RoboDK station: kr30 cnc 040719 5.rdk

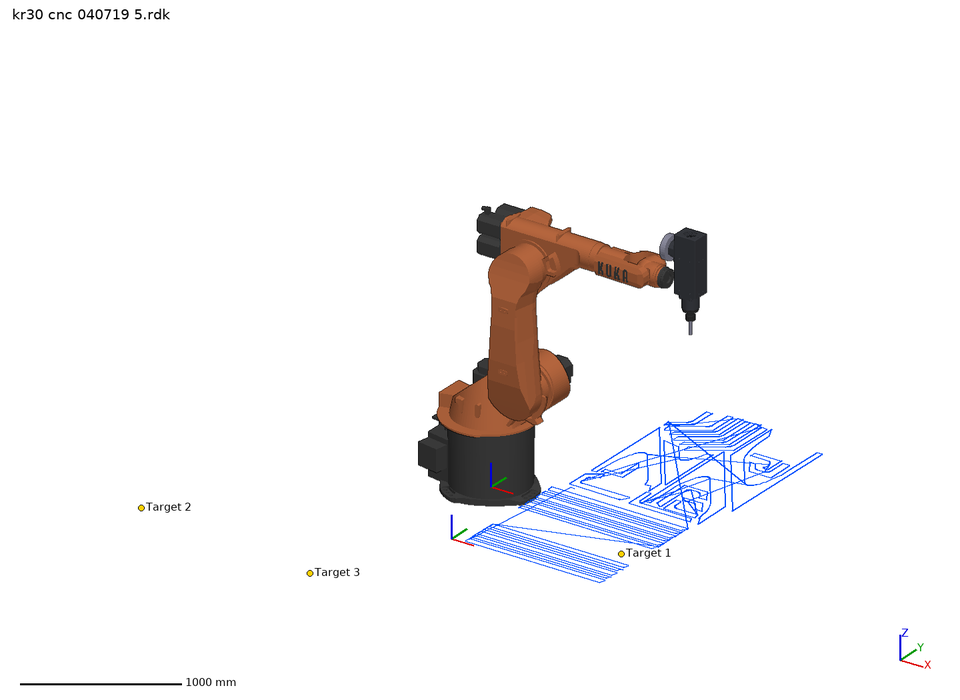
[picture v0: the station drawn from its stored meshes, robots at their saved joint values, targets as dots, program paths as lines]
Station kr30 cnc 040719 5. Poses are relative to the parent item; angles as X-Y-Z fixed-axis rotations.
  - frame KUKA KR 30 HA Base at (0, 0, 0) mm
    - robot KUKA KR 30 HA: 6 axes, payload 30 kg, reach 2033 mm, repeatability 0.05 mm, weight 665 kg
        modified DH rows (alpha deg, a mm, theta deg, d mm): 0, 0, 0, 815; -90, 350, 0, 0; 0, 850, -90, 0; -90, 145, 0, 820; 90, 0, 0, 0; -90, 0, 180, 170
        joint limits [-185, -135, -120, -350, -119, -350] to [185, 35, 158, 350, 119, 350]; home [0, -90, 90, 0, 0, 0]; saved at [0, -90, 90, 0, 0, 0]
      - tool 1/2" End Mill TCP, TCP at (337.71, -2.2, 160.57) mm, size 692.9 x 170 x 256 mm
    - frame Reference Rhino at (538.65, -1191.99, 269.68) mm
      - target Target 1 (Cartesian target) at (994.45, 406.4, 10) mm, rotated rx 0 ry 90 rz -60.43 deg; joints [16.304, -19.243, 71.371, -50.859, -63.853, 28.433] of KUKA KR 30 HA
      - target Target 2 (Cartesian target) at (-1810.84, -765.32, 10.08) mm, rotated rx 49.23 ry 89.99 rz -110.09 deg; joints [109.009, -5.295, 40.673, -64.339, -58.629, 47.297] of KUKA KR 30 HA
      - target Target 3 (Cartesian target) at (-425.52, -920.6, 10.08) mm, rotated rx 49.23 ry 89.99 rz -69.31 deg; joints [71.775, -8.447, 47.414, -59.408, -57.827, 42.008] of KUKA KR 30 HA
      - object RhinoPart at (0, 0, 0) mm
  - machining project RhinoPart Settings: C:/Users/Julian Ramirez.DESKTOP-JVDE542/Desktop/ELMER SHEET 1 TEST 3.nc | rotX(0) | rotY(270)*rotX(-65)
  - object box at (500, 500, 500) mm, size 250 x 250 x 250 mm, geometry from box.sld
  - program RhinoPart (549 instructions, listed below)
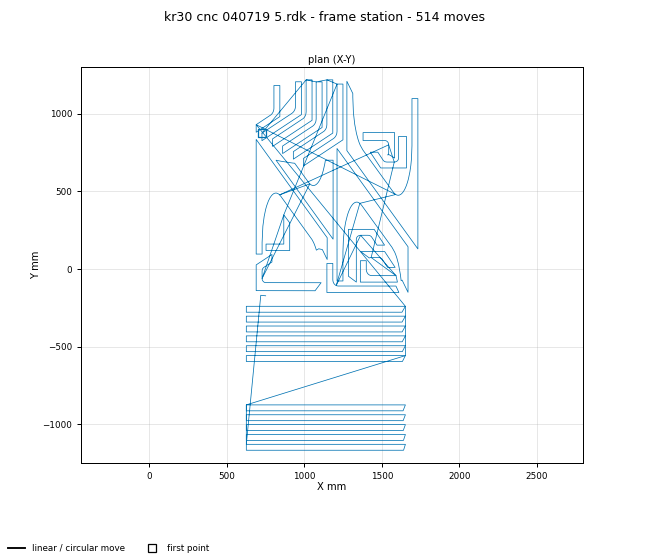
[picture p0: tool path of kr30 cnc 040719 5.rdk in frame station, 514 of 514 moves have a stored position in this frame; points joined in program order, loops and branches not executed]

--- program RhinoPart (robot KUKA KR 30 HA) ---
  Smooth(1)
  Set Ref.: Reference Rhino
  Set Tool: 1/2" End Mill TCP
  Show 1/2" End Mill TCP
  Set speed (2000.0 mm/s)
  MoveJ 1 to (189.6, 2067.69, 0) mm, rotated rx 0 ry 90 rz 29.57 deg; joints [-58.394, -46.833, 153.246, -29.84, -104.333, -8.083]
  MoveL 2 to (189.6, 2067.69, 0) mm, rotated rx 0 ry 90 rz 29.57 deg; joints [-58.394, -46.833, 153.246, -29.84, -104.333, -8.083]
  MoveL 3 to (189.6, 2067.69, 0) mm, rotated rx 0 ry 90 rz 29.57 deg; joints [-58.394, -46.833, 153.246, -29.84, -104.333, -8.083]
  Set speed (60.0 mm/s)
  MoveL 4 to (189.6, 2019.15, 0) mm, rotated rx 0 ry 90 rz 29.57 deg; joints [-56.567, -46.166, 155.923, -28.426, -107.53, -9.26]
  MoveL 5 to (443.6, 2187.03, 0) mm, rotated rx 0 ry 90 rz 29.57 deg; joints [-50.243, -46.091, 136.083, -20.671, -89.992, 0.003]
  MoveL 6 to (443.6, 2398.44, 0) mm, rotated rx 0 ry 90 rz 29.57 deg; joints [-56.43, -42.72, 123.102, -27.187, -81.428, 4.378]
  MoveL 7 to (405.5, 2398.44, 0) mm, rotated rx 0 ry 90 rz 29.57 deg; joints [-57.905, -43.217, 124.737, -28.597, -82.542, 4.047]
  MoveL 8 to (405.5, 2241.51, 0) mm, rotated rx 0 ry 90 rz 29.57 deg; joints [-53.573, -45.796, 134.651, -24.006, -88.954, 0.466]
  MoveL 9 to (405.1, 2234.61, 0) mm, rotated rx 0 ry 90 rz 29.57 deg; joints [-53.376, -45.887, 135.079, -23.806, -89.261, 0.326]
  MoveL 10 to (403.91, 2227.8, 0) mm, rotated rx 0 ry 90 rz 29.57 deg; joints [-53.213, -45.981, 135.535, -23.642, -89.591, 0.179]
  MoveL 11 to (401.94, 2221.18, 0) mm, rotated rx 0 ry 90 rz 29.57 deg; joints [-53.087, -46.077, 136.012, -23.515, -89.941, 0.026]
  MoveL 12 to (399.2, 2214.83, 0) mm, rotated rx 0 ry 90 rz 29.57 deg; joints [-53.001, -46.174, 136.507, -23.43, -90.305, -0.132]
  MoveL 13 to (395.69, 2208.84, 0) mm, rotated rx 0 ry 90 rz 29.57 deg; joints [-52.958, -46.27, 137.012, -23.388, -90.682, -0.295]
  MoveL 14 to (391.47, 2203.34, 0) mm, rotated rx 0 ry 90 rz 29.57 deg; joints [-52.961, -46.362, 137.518, -23.394, -91.061, -0.459]
  MoveL 15 to (386.58, 2198.44, 0) mm, rotated rx 0 ry 90 rz 29.57 deg; joints [-53.013, -46.45, 138.017, -23.449, -91.438, -0.624]
  MoveL 16 to (383.89, 2196.24, 0) mm, rotated rx 0 ry 90 rz 29.57 deg; joints [-53.057, -46.492, 138.263, -23.496, -91.624, -0.706]
  MoveL 17 to (381.06, 2194.23, 0) mm, rotated rx 0 ry 90 rz 29.57 deg; joints [-53.115, -46.533, 138.503, -23.556, -91.807, -0.788]
  MoveL 18 to (189.6, 2067.69, 0) mm, rotated rx 0 ry 90 rz 29.57 deg; joints [-58.394, -46.833, 153.246, -29.84, -104.333, -8.083]
  MoveL 19 to (474.07, 2410.87, 0) mm, rotated rx 0 ry 90 rz 29.57 deg; joints [-55.602, -42.027, 120.911, -26.461, -80.024, 4.928]
  Set speed (60.0 mm/s)
  MoveL 20 to (512.17, 2410.87, 0) mm, rotated rx 0 ry 90 rz 29.57 deg; joints [-54.221, -41.445, 119.132, -25.158, -78.824, 5.201]
  MoveL 21 to (512.17, 2150.2, 0) mm, rotated rx 0 ry 90 rz 29.57 deg; joints [-46.277, -45.815, 134.74, -16.708, -88.97, 0.309]
  MoveL 22 to (258.17, 1982.32, 0) mm, rotated rx 0 ry 90 rz 29.57 deg; joints [-51.067, -46.373, 155.224, -22.594, -107.496, -7.131]
  MoveL 23 to (258.17, 2030.85, 0) mm, rotated rx 0 ry 90 rz 29.57 deg; joints [-53.13, -46.929, 152.707, -24.376, -104.433, -6.444]
  MoveL 24 to (449.63, 2157.39, 0) mm, rotated rx 0 ry 90 rz 29.57 deg; joints [-48.975, -46.35, 137.45, -19.406, -91.038, -0.366]
  MoveL 25 to (455.15, 2161.61, 0) mm, rotated rx 0 ry 90 rz 29.57 deg; joints [-48.9, -46.258, 136.952, -19.33, -90.655, -0.23]
  MoveL 26 to (460.04, 2166.51, 0) mm, rotated rx 0 ry 90 rz 29.57 deg; joints [-48.876, -46.162, 136.446, -19.304, -90.268, -0.094]
  MoveL 27 to (464.26, 2172, 0) mm, rotated rx 0 ry 90 rz 29.57 deg; joints [-48.898, -46.062, 135.938, -19.327, -89.883, 0.041]
  MoveL 28 to (467.77, 2178, 0) mm, rotated rx 0 ry 90 rz 29.57 deg; joints [-48.966, -45.961, 135.435, -19.395, -89.504, 0.175]
  MoveL 29 to (470.51, 2184.35, 0) mm, rotated rx 0 ry 90 rz 29.57 deg; joints [-49.076, -45.859, 134.947, -19.506, -89.14, 0.305]
  MoveL 30 to (472.48, 2190.97, 0) mm, rotated rx 0 ry 90 rz 29.57 deg; joints [-49.223, -45.76, 134.48, -19.656, -88.795, 0.43]
  MoveL 31 to (474.07, 2204.68, 0) mm, rotated rx 0 ry 90 rz 29.57 deg; joints [-49.621, -45.572, 133.629, -20.06, -88.175, 0.666]
  MoveL 32 to (474.07, 2410.87, 0) mm, rotated rx 0 ry 90 rz 29.57 deg; joints [-55.602, -42.027, 120.911, -26.461, -80.024, 4.928]
  MoveL 33 to (538.73, 2397.73, 0) mm, rotated rx 0 ry 90 rz 29.57 deg; joints [-52.941, -41.304, 118.707, -23.882, -78.452, 5.065]
  Set speed (60.0 mm/s)
  MoveL 34 to (538.73, 2158.69, 0) mm, rotated rx 0 ry 90 rz 29.57 deg; joints [-45.6, -45.407, 132.909, -16.043, -87.598, 0.69]
  MoveL 35 to (537.14, 2144.98, 0) mm, rotated rx 0 ry 90 rz 29.57 deg; joints [-45.166, -45.593, 133.721, -15.602, -88.197, 0.503]
  MoveL 36 to (535.17, 2138.36, 0) mm, rotated rx 0 ry 90 rz 29.57 deg; joints [-44.997, -45.693, 134.174, -15.431, -88.536, 0.404]
  MoveL 37 to (532.43, 2132.01, 0) mm, rotated rx 0 ry 90 rz 29.57 deg; joints [-44.865, -45.797, 134.652, -15.296, -88.896, 0.302]
  MoveL 38 to (528.92, 2126.02, 0) mm, rotated rx 0 ry 90 rz 29.57 deg; joints [-44.772, -45.902, 135.149, -15.202, -89.274, 0.197]
  MoveL 39 to (524.7, 2120.53, 0) mm, rotated rx 0 ry 90 rz 29.57 deg; joints [-44.723, -46.006, 135.656, -15.152, -89.662, 0.091]
  MoveL 40 to (519.81, 2115.63, 0) mm, rotated rx 0 ry 90 rz 29.57 deg; joints [-44.721, -46.107, 136.165, -15.15, -90.056, -0.015]
  MoveL 41 to (514.29, 2111.41, 0) mm, rotated rx 0 ry 90 rz 29.57 deg; joints [-44.769, -46.205, 136.671, -15.197, -90.45, -0.122]
  MoveL 42 to (322.83, 1984.87, 0) mm, rotated rx 0 ry 90 rz 29.57 deg; joints [-47.793, -46.99, 152.328, -18.848, -104.552, -4.902]
  MoveL 43 to (322.83, 1936.34, 0) mm, rotated rx 0 ry 90 rz 29.57 deg; joints [-45.507, -46.523, 154.657, -16.723, -107.414, -5.138]
  MoveL 44 to (576.83, 2104.21, 0) mm, rotated rx 0 ry 90 rz 29.57 deg; joints [-42.246, -45.584, 133.683, -12.682, -88.145, 0.417]
  MoveL 45 to (576.83, 2397.73, 0) mm, rotated rx 0 ry 90 rz 29.57 deg; joints [-51.633, -40.652, 116.785, -22.658, -77.166, 5.298]
  MoveL 46 to (538.73, 2397.73, 0) mm, rotated rx 0 ry 90 rz 29.57 deg; joints [-52.941, -41.304, 118.707, -23.882, -78.452, 5.065]
  MoveL 47 to (607.72, 2410.87, 0) mm, rotated rx 0 ry 90 rz 29.57 deg; joints [-50.958, -39.788, 114.308, -22.115, -75.61, 5.767]
  Set speed (60.0 mm/s)
  MoveL 48 to (645.82, 2410.87, 0) mm, rotated rx 0 ry 90 rz 29.57 deg; joints [-49.734, -39.045, 112.237, -20.986, -74.25, 5.944]
  MoveL 49 to (645.82, 2068.09, 0) mm, rotated rx 0 ry 90 rz 29.57 deg; joints [-38.589, -45.07, 131.497, -9.034, -86.471, 0.561]
  MoveL 50 to (391.82, 1900.22, 0) mm, rotated rx 0 ry 90 rz 29.57 deg; joints [-40.437, -46.886, 152.953, -11.296, -105.771, -3.108]
  MoveL 51 to (391.82, 1948.75, 0) mm, rotated rx 0 ry 90 rz 29.57 deg; joints [-42.855, -47.182, 150.8, -13.654, -103.247, -3.186]
  MoveL 52 to (583.27, 2075.29, 0) mm, rotated rx 0 ry 90 rz 29.57 deg; joints [-40.908, -45.818, 134.752, -11.339, -88.955, 0.21]
  MoveL 53 to (588.8, 2079.51, 0) mm, rotated rx 0 ry 90 rz 29.57 deg; joints [-40.886, -45.707, 134.237, -11.318, -88.558, 0.289]
  MoveL 54 to (593.69, 2084.41, 0) mm, rotated rx 0 ry 90 rz 29.57 deg; joints [-40.912, -45.593, 133.723, -11.347, -88.166, 0.368]
  MoveL 55 to (597.91, 2089.9, 0) mm, rotated rx 0 ry 90 rz 29.57 deg; joints [-40.983, -45.478, 133.216, -11.42, -87.782, 0.448]
  MoveL 56 to (601.42, 2095.89, 0) mm, rotated rx 0 ry 90 rz 29.57 deg; joints [-41.096, -45.364, 132.723, -11.536, -87.412, 0.528]
  MoveL 57 to (604.16, 2102.24, 0) mm, rotated rx 0 ry 90 rz 29.57 deg; joints [-41.246, -45.253, 132.253, -11.69, -87.063, 0.608]
  MoveL 58 to (606.13, 2108.87, 0) mm, rotated rx 0 ry 90 rz 29.57 deg; joints [-41.431, -45.147, 131.813, -11.879, -86.737, 0.686]
  MoveL 59 to (607.72, 2122.58, 0) mm, rotated rx 0 ry 90 rz 29.57 deg; joints [-41.89, -44.955, 131.034, -12.346, -86.17, 0.838]
  MoveL 60 to (607.72, 2410.87, 0) mm, rotated rx 0 ry 90 rz 29.57 deg; joints [-50.958, -39.788, 114.308, -22.115, -75.61, 5.767]
  MoveL 61 to (673.1, 2383.75, 0) mm, rotated rx 0 ry 90 rz 29.57 deg; joints [-48.146, -39.124, 112.454, -19.33, -74.222, 5.448]
  Set speed (60.0 mm/s)
  MoveL 62 to (673.1, 2079.03, 0) mm, rotated rx 0 ry 90 rz 29.57 deg; joints [-38.176, -44.522, 129.354, -8.639, -84.89, 0.775]
  MoveL 63 to (671.52, 2065.32, 0) mm, rotated rx 0 ry 90 rz 29.57 deg; joints [-37.693, -44.715, 130.093, -8.148, -85.424, 0.654]
  MoveL 64 to (669.55, 2058.7, 0) mm, rotated rx 0 ry 90 rz 29.57 deg; joints [-37.494, -44.825, 130.519, -7.945, -85.735, 0.595]
  MoveL 65 to (666.8, 2052.35, 0) mm, rotated rx 0 ry 90 rz 29.57 deg; joints [-37.327, -44.941, 130.977, -7.773, -86.073, 0.536]
  MoveL 66 to (663.29, 2046.36, 0) mm, rotated rx 0 ry 90 rz 29.57 deg; joints [-37.195, -45.061, 131.463, -7.638, -86.434, 0.478]
  MoveL 67 to (659.07, 2040.86, 0) mm, rotated rx 0 ry 90 rz 29.57 deg; joints [-37.103, -45.184, 131.967, -7.543, -86.811, 0.422]
  MoveL 68 to (654.18, 2035.96, 0) mm, rotated rx 0 ry 90 rz 29.57 deg; joints [-37.055, -45.308, 132.483, -7.492, -87.2, 0.368]
  MoveL 69 to (648.66, 2031.74, 0) mm, rotated rx 0 ry 90 rz 29.57 deg; joints [-37.053, -45.429, 133.004, -7.488, -87.596, 0.316]
  MoveL 70 to (457.2, 1905.21, 0) mm, rotated rx 0 ry 90 rz 29.57 deg; joints [-37.971, -47.293, 149.341, -8.586, -101.917, -1.786]
  MoveL 71 to (457.2, 1856.67, 0) mm, rotated rx 0 ry 90 rz 29.57 deg; joints [-35.445, -47.128, 151.299, -6.056, -104.096, -1.48]
  MoveL 72 to (711.2, 2024.55, 0) mm, rotated rx 0 ry 90 rz 29.57 deg; joints [-34.93, -44.559, 129.495, -5.379, -84.958, 0.474]
  MoveL 73 to (711.2, 2383.75, 0) mm, rotated rx 0 ry 90 rz 29.57 deg; joints [-46.992, -38.31, 110.233, -18.266, -72.779, 5.581]
  MoveL 74 to (673.1, 2383.75, 0) mm, rotated rx 0 ry 90 rz 29.57 deg; joints [-48.146, -39.124, 112.454, -19.33, -74.222, 5.448]
  MoveL 75 to (330.2, 1541.24, 0) mm, rotated rx 180 ry 60 rz -150.43 deg; joints [-20.955, -60.967, 157.047, 8.164, -66.015, 0.995]
  Set speed (60.0 mm/s)
  MoveL 76 to (365.54, 1493.75, 0) mm, rotated rx -180 ry 60 rz -150.43 deg; joints [-17.055, -60.795, 155.789, 11.964, -64.88, 1.194]
  MoveL 77 to (368.3, 1490.21, 0) mm, rotated rx -180 ry 60 rz -150.43 deg; joints [-16.768, -60.778, 155.676, 12.248, -64.781, 1.198]
  MoveL 78 to (368.3, 1311.73, 0) mm, rotated rx -180 ry 60 rz -150.43 deg; joints [-4.531, -61.072, 157.995, 23.596, -66.311, 3.194]
  MoveL 79 to (215.9, 1311.73, 0) mm, rotated rx -180 ry 30 rz -150.43 deg; joints [-12.047, -59.926, 152.531, 16.276, -32.492, 1.46]
  MoveL 80 to (215.9, 1353.22, 0) mm, rotated rx -180 ry 40 rz -150.43 deg; joints [-13.186, -62.573, 157.529, 14.92, -44.772, 1.983]
  MoveL 81 to (330.2, 1353.22, 0) mm, rotated rx -180 ry 50 rz -150.43 deg; joints [-9.855, -62.245, 155.167, 18.943, -52.758, 1.238]
  MoveL 82 to (330.2, 1541.24, 0) mm, rotated rx -180 ry 60 rz -150.43 deg; joints [-20.955, -60.967, 157.047, 8.164, -66.015, 0.995]
  MoveL 83 to (190.5, 1131.98, 0) mm, rotated rx -180 ry 30 rz -150.43 deg; joints [-0.319, -60.475, 155.694, 25.458, -34.639, 4.485]
  Set speed (60.0 mm/s)
  MoveL 84 to (190.5, 1180.23, 0) mm, rotated rx -180 ry 30 rz -150.43 deg; joints [-3.61, -60.458, 155.578, 22.631, -34.669, 3.938]
  MoveL 85 to (191.3, 1187.11, 0) mm, rotated rx -180 ry 30 rz -150.43 deg; joints [-4.074, -60.445, 155.489, 22.265, -34.615, 3.82]
  MoveL 86 to (192.29, 1190.42, 0) mm, rotated rx -180 ry 30 rz -150.43 deg; joints [-4.294, -60.432, 155.403, 22.112, -34.554, 3.74]
  MoveL 87 to (193.65, 1193.58, 0) mm, rotated rx -180 ry 30 rz -150.43 deg; joints [-4.501, -60.415, 155.291, 21.982, -34.472, 3.648]
  MoveL 88 to (195.39, 1196.56, 0) mm, rotated rx -180 ry 30 rz -150.43 deg; joints [-4.692, -60.394, 155.152, 21.877, -34.369, 3.544]
  MoveL 89 to (197.49, 1199.29, 0) mm, rotated rx -180 ry 30 rz -150.43 deg; joints [-4.865, -60.369, 154.99, 21.799, -34.247, 3.43]
  MoveL 90 to (199.93, 1201.75, 0) mm, rotated rx -180 ry 30 rz -150.43 deg; joints [-5.016, -60.339, 154.803, 21.751, -34.106, 3.307]
  MoveL 91 to (202.72, 1203.88, 0) mm, rotated rx -180 ry 30 rz -150.43 deg; joints [-5.142, -60.305, 154.595, 21.735, -33.947, 3.175]
  MoveL 92 to (254, 1237.77, 0) mm, rotated rx -180 ry 40 rz -150.43 deg; joints [-4.845, -62.336, 156.153, 22.996, -43.491, 2.319]
  MoveL 93 to (254, 1286.3, 0) mm, rotated rx -180 ry 40 rz -150.43 deg; joints [-8.144, -62.263, 155.766, 20.032, -43.277, 1.866]
  MoveL 94 to (152.4, 1219.15, 0) mm, rotated rx -180 ry 30 rz -150.43 deg; joints [-6.544, -60.743, 157.989, 19.072, -36.768, 4.728]
  MoveL 95 to (152.4, 1053.37, 0) mm, rotated rx -180 ry 20 rz -150.43 deg; joints [2.369, -56.869, 153.192, 24.779, -25.576, 7.756]
  MoveL 96 to (520.7, 1053.37, 0) mm, rotated rx 0 ry 90 rz 29.57 deg; joints [21.258, -46.671, 154.029, 52.131, -100.861, 13.621]
  MoveL 97 to (523.39, 1053.29, 0) mm, rotated rx 0 ry 90 rz 29.57 deg; joints [21.196, -46.708, 153.862, 52.038, -100.751, 13.446]
  MoveL 98 to (526.09, 1053.06, 0) mm, rotated rx 0 ry 90 rz 29.57 deg; joints [21.144, -46.744, 153.691, 51.956, -100.635, 13.271]
  MoveL 99 to (528.75, 1052.67, 0) mm, rotated rx 0 ry 90 rz 29.57 deg; joints [21.102, -46.78, 153.518, 51.884, -100.516, 13.096]
  MoveL 100 to (531.38, 1052.13, 0) mm, rotated rx 0 ry 90 rz 29.57 deg; joints [21.072, -46.814, 153.343, 51.824, -100.394, 12.924]
  MoveL 101 to (570.41, 1104.33, 0) mm, rotated rx 0 ry 90 rz 29.57 deg; joints [16.876, -47.035, 152.019, 47.436, -100.261, 10.977]
  MoveL 102 to (215.9, 1104.33, 0) mm, rotated rx 180 ry 30 rz -150.43 deg; joints [1.524, -60.184, 153.886, 28.122, -33.22, 3.49]
  MoveL 103 to (210.71, 1104.91, 0) mm, rotated rx -180 ry 30 rz -150.43 deg; joints [1.494, -60.248, 154.253, 27.879, -33.489, 3.745]
  MoveL 104 to (208.23, 1105.62, 0) mm, rotated rx -180 ry 30 rz -150.43 deg; joints [1.451, -60.278, 154.429, 27.738, -33.619, 3.864]
  MoveL 105 to (205.85, 1106.58, 0) mm, rotated rx -180 ry 30 rz -150.43 deg; joints [1.391, -60.306, 154.599, 27.585, -33.746, 3.975]
  MoveL 106 to (203.58, 1107.8, 0) mm, rotated rx -180 ry 30 rz -150.43 deg; joints [1.313, -60.332, 154.76, 27.421, -33.869, 4.078]
  MoveL 107 to (201.44, 1109.25, 0) mm, rotated rx -180 ry 30 rz -150.43 deg; joints [1.218, -60.357, 154.913, 27.25, -33.986, 4.171]
  MoveL 108 to (199.45, 1110.91, 0) mm, rotated rx -180 ry 30 rz -150.43 deg; joints [1.109, -60.379, 155.056, 27.071, -34.097, 4.255]
  MoveL 109 to (197.61, 1112.79, 0) mm, rotated rx -180 ry 30 rz -150.43 deg; joints [0.984, -60.4, 155.187, 26.886, -34.201, 4.329]
  MoveL 110 to (195.97, 1114.84, 0) mm, rotated rx -180 ry 30 rz -150.43 deg; joints [0.847, -60.418, 155.305, 26.698, -34.295, 4.39]
  MoveL 111 to (194.53, 1117.03, 0) mm, rotated rx -180 ry 30 rz -150.43 deg; joints [0.7, -60.433, 155.407, 26.511, -34.379, 4.44]
  MoveL 112 to (192.31, 1121.74, 0) mm, rotated rx 180 ry 30 rz -150.43 deg; joints [0.38, -60.456, 155.567, 26.141, -34.513, 4.502]
  MoveL 113 to (190.96, 1126.77, 0) mm, rotated rx -180 ry 30 rz -150.43 deg; joints [0.037, -60.47, 155.663, 25.787, -34.601, 4.516]
  MoveL 114 to (190.5, 1131.98, 0) mm, rotated rx -180 ry 30 rz -150.43 deg; joints [-0.319, -60.475, 155.694, 25.458, -34.639, 4.485]
  MoveL 115 to (497.79, 1740.88, 0) mm, rotated rx -180 ry 80 rz -150.43 deg; joints [-27.553, -52.725, 149.919, 1.99, -87.19, 0.253]
  Set speed (60.0 mm/s)
  MoveL 116 to (502.27, 1737.01, 0) mm, rotated rx 0 ry 90 rz 29.57 deg; joints [-27.028, -46.901, 152.872, 2.646, -105.955, 0.728]
  MoveL 117 to (506.69, 1734.05, 0) mm, rotated rx 0 ry 90 rz 29.57 deg; joints [-26.714, -46.93, 152.699, 2.969, -105.749, 0.807]
  MoveL 118 to (511.04, 1731.95, 0) mm, rotated rx 0 ry 90 rz 29.57 deg; joints [-26.455, -46.962, 152.503, 3.234, -105.517, 0.866]
  MoveL 119 to (515.31, 1730.65, 0) mm, rotated rx 0 ry 90 rz 29.57 deg; joints [-26.249, -46.996, 152.287, 3.444, -105.264, 0.908]
  MoveL 120 to (519.5, 1730.11, 0) mm, rotated rx 0 ry 90 rz 29.57 deg; joints [-26.093, -47.031, 152.052, 3.601, -104.993, 0.933]
  MoveL 121 to (523.61, 1730.27, 0) mm, rotated rx 0 ry 90 rz 29.57 deg; joints [-25.983, -47.065, 151.801, 3.711, -104.706, 0.943]
  MoveL 122 to (527.62, 1731.09, 0) mm, rotated rx 0 ry 90 rz 29.57 deg; joints [-25.915, -47.1, 151.536, 3.775, -104.406, 0.941]
  MoveL 123 to (531.52, 1732.52, 0) mm, rotated rx 0 ry 90 rz 29.57 deg; joints [-25.887, -47.133, 151.259, 3.799, -104.097, 0.926]
  MoveL 124 to (535.31, 1734.5, 0) mm, rotated rx 0 ry 90 rz 29.57 deg; joints [-25.896, -47.164, 150.972, 3.785, -103.779, 0.903]
  MoveL 125 to (538.98, 1736.99, 0) mm, rotated rx 0 ry 90 rz 29.57 deg; joints [-25.937, -47.194, 150.677, 3.737, -103.455, 0.871]
  MoveL 126 to (542.53, 1739.94, 0) mm, rotated rx 0 ry 90 rz 29.57 deg; joints [-26.009, -47.221, 150.375, 3.659, -103.128, 0.832]
  MoveL 127 to (545.93, 1743.29, 0) mm, rotated rx 0 ry 90 rz 29.57 deg; joints [-26.107, -47.246, 150.069, 3.553, -102.799, 0.788]
  MoveL 128 to (552.31, 1751, 0) mm, rotated rx 0 ry 90 rz 29.57 deg; joints [-26.37, -47.287, 149.45, 3.274, -102.144, 0.69]
  MoveL 129 to (557.85, 1759.34, 0) mm, rotated rx 0 ry 90 rz 29.57 deg; joints [-26.688, -47.315, 148.86, 2.943, -101.53, 0.589]
  MoveL 130 to (562.91, 1768.41, 0) mm, rotated rx 0 ry 90 rz 29.57 deg; joints [-27.054, -47.334, 148.271, 2.564, -100.927, 0.486]
  MoveL 131 to (567.51, 1777.97, 0) mm, rotated rx 0 ry 90 rz 29.57 deg; joints [-27.453, -47.343, 147.691, 2.154, -100.341, 0.387]
  MoveL 132 to (576.13, 1799.75, 0) mm, rotated rx 0 ry 90 rz 29.57 deg; joints [-28.39, -47.334, 146.463, 1.197, -99.127, 0.19]
  MoveL 133 to (584.02, 1825.23, 0) mm, rotated rx 0 ry 90 rz 29.57 deg; joints [-29.506, -47.284, 145.126, 0.067, -97.843, 0.009]
  MoveL 134 to (593.39, 1865.46, 0) mm, rotated rx 0 ry 90 rz 29.57 deg; joints [-31.271, -47.139, 143.131, -1.709, -95.989, -0.178]
  MoveL 135 to (598.13, 1892.37, 0) mm, rotated rx 0 ry 90 rz 29.57 deg; joints [-32.442, -47.005, 141.839, -2.881, -94.828, -0.243]
  MoveL 136 to (609.6, 1893.44, 0) mm, rotated rx 0 ry 90 rz 29.57 deg; joints [-32.146, -46.916, 141.107, -2.581, -94.186, -0.189]
  MoveL 137 to (647.7, 1893.44, 0) mm, rotated rx 0 ry 90 rz 29.57 deg; joints [-31.037, -46.577, 138.772, -1.467, -92.195, -0.056]
  MoveL 138 to (647.7, 1384.85, 0) mm, rotated rx 0 ry 90 rz 29.57 deg; joints [-2.018, -47.297, 149.263, 28.074, -100.592, 5.599]
  MoveL 139 to (280.37, 1893.44, 0) mm, rotated rx -180 ry 80 rz -150.43 deg; joints [-44.299, -52.692, 155.935, -14.517, -92.817, -3.343]
  MoveL 140 to (309.91, 1887.14, 0) mm, rotated rx 0 ry 90 rz 29.57 deg; joints [-43.636, -45.609, 157.481, -15.108, -111.184, -5.572]
  MoveL 141 to (385.37, 1875.31, 0) mm, rotated rx 0 ry 90 rz 29.57 deg; joints [-39.408, -46.602, 154.332, -10.317, -107.461, -3.126]
  MoveL 142 to (400.34, 1873.88, 0) mm, rotated rx 0 ry 90 rz 29.57 deg; joints [-38.679, -46.757, 153.628, -9.509, -106.651, -2.748]
  MoveL 143 to (488.7, 1751.54, 0) mm, rotated rx 0 ry 90 rz 29.57 deg; joints [-28.332, -46.837, 153.22, 1.292, -106.379, 0.364]
  MoveL 144 to (493.27, 1745.7, 0) mm, rotated rx 0 ry 90 rz 29.57 deg; joints [-27.835, -46.853, 153.135, 1.809, -106.274, 0.507]
  MoveL 145 to (497.79, 1740.88, 0) mm, rotated rx 0 ry 90 rz 29.57 deg; joints [-27.401, -46.875, 153.018, 2.26, -106.131, 0.628]
  MoveL 146 to (303.35, 1670.14, 0) mm, rotated rx -180 ry 60 rz -150.43 deg; joints [-29.742, -60.649, 154.872, -0.164, -64.222, -0.014]
  Set speed (60.0 mm/s)
  MoveL 147 to (307.39, 1665.7, 0) mm, rotated rx -180 ry 60 rz -150.43 deg; joints [-29.348, -60.634, 154.778, 0.215, -64.144, 0.018]
  MoveL 148 to (311.4, 1660.54, 0) mm, rotated rx -180 ry 60 rz -150.43 deg; joints [-28.914, -60.622, 154.708, 0.633, -64.086, 0.052]
  MoveL 149 to (511.79, 1382.48, 0) mm, rotated rx -180 ry 80 rz -150.43 deg; joints [-4.246, -52.699, 155.869, 24.929, -91.933, 5.596]
  MoveL 150 to (516.77, 1373.81, 0) mm, rotated rx 0 ry 90 rz 29.57 deg; joints [-1.538, -45.433, 157.901, 29.951, -109.714, 11]
  MoveL 151 to (521.42, 1364.56, 0) mm, rotated rx 0 ry 90 rz 29.57 deg; joints [-0.842, -45.553, 157.618, 30.603, -109.233, 11.025]
  MoveL 152 to (525.76, 1354.87, 0) mm, rotated rx 0 ry 90 rz 29.57 deg; joints [-0.122, -45.662, 157.346, 31.284, -108.769, 11.062]
  MoveL 153 to (533.5, 1334.64, 0) mm, rotated rx 0 ry 90 rz 29.57 deg; joints [1.359, -45.856, 156.837, 32.691, -107.887, 11.151]
  MoveL 154 to (540.04, 1314.08, 0) mm, rotated rx 0 ry 90 rz 29.57 deg; joints [2.836, -46.02, 156.369, 34.1, -107.072, 11.242]
  MoveL 155 to (555.23, 1322.96, 0) mm, rotated rx 0 ry 90 rz 29.57 deg; joints [2.152, -46.319, 155.412, 33.192, -106.155, 10.316]
  MoveL 156 to (561.07, 1321.73, 0) mm, rotated rx 0 ry 90 rz 29.57 deg; joints [2.223, -46.426, 155.029, 33.188, -105.732, 10.057]
  MoveL 157 to (578.58, 1317.86, 0) mm, rotated rx 0 ry 90 rz 29.57 deg; joints [2.444, -46.706, 153.873, 33.201, -104.494, 9.301]
  MoveL 158 to (609.6, 1253.88, 0) mm, rotated rx 0 ry 90 rz 29.57 deg; joints [6.592, -47.106, 151.485, 37.037, -101.566, 8.603]
  MoveL 159 to (609.6, 1394.22, 0) mm, rotated rx 0 ry 90 rz 29.57 deg; joints [-2.73, -47.065, 151.802, 27.621, -103.119, 6.773]
  MoveL 160 to (152.4, 2027.23, 0) mm, rotated rx 180 ry 70 rz -150.43 deg; joints [-54.922, -56.98, 150.659, -24.834, -73.332, -1.643]
  MoveL 161 to (152.4, 1288.87, 0) mm, rotated rx 180 ry 20 rz -150.43 deg; joints [-12.956, -56.684, 151.653, 13.483, -24.8, 3.385]
  MoveL 162 to (190.5, 1288.87, 0) mm, rotated rx -180 ry 30 rz -150.43 deg; joints [-10.903, -60.308, 154.611, 16.586, -34.102, 2.455]
  MoveL 163 to (190.5, 1362.91, 0) mm, rotated rx -180 ry 30 rz -150.43 deg; joints [-15.691, -60.096, 153.409, 12.646, -33.224, 1.45]
  MoveL 164 to (195.47, 1468.11, 0) mm, rotated rx -180 ry 40 rz -150.43 deg; joints [-21.259, -62.401, 156.508, 7.678, -44.067, 0.853]
  MoveL 165 to (203.82, 1530.87, 0) mm, rotated rx -180 ry 40 rz -150.43 deg; joints [-24.948, -61.945, 154.226, 4.417, -42.274, 0.273]
  MoveL 166 to (213.36, 1576.46, 0) mm, rotated rx -180 ry 40 rz -150.43 deg; joints [-27.349, -61.467, 152.189, 2.19, -40.722, 0.043]
  MoveL 167 to (219.68, 1599.23, 0) mm, rotated rx -180 ry 50 rz -150.43 deg; joints [-28.331, -62.572, 156.878, 1.17, -54.305, 0.115]
  MoveL 168 to (227.14, 1620.99, 0) mm, rotated rx -180 ry 50 rz -150.43 deg; joints [-29.394, -62.348, 155.679, 0.17, -53.331, 0.013]
  MoveL 169 to (231.16, 1630.88, 0) mm, rotated rx -180 ry 50 rz -150.43 deg; joints [-29.842, -62.228, 155.087, -0.259, -52.859, -0.017]
  MoveL 170 to (235.75, 1640.83, 0) mm, rotated rx -180 ry 50 rz -150.43 deg; joints [-30.265, -62.093, 154.453, -0.671, -52.36, -0.036]
  MoveL 171 to (240.92, 1650.5, 0) mm, rotated rx -180 ry 50 rz -150.43 deg; joints [-30.644, -61.945, 153.79, -1.045, -51.845, -0.044]
  MoveL 172 to (246.67, 1659.52, 0) mm, rotated rx -180 ry 50 rz -150.43 deg; joints [-30.959, -61.786, 153.111, -1.362, -51.324, -0.041]
  MoveL 173 to (250.51, 1664.62, 0) mm, rotated rx -180 ry 50 rz -150.43 deg; joints [-31.115, -61.684, 152.689, -1.521, -51.005, -0.035]
  MoveL 174 to (254.42, 1669.07, 0) mm, rotated rx -180 ry 60 rz -150.43 deg; joints [-31.397, -61.058, 157.861, -1.72, -66.799, -0.235]
  MoveL 175 to (258.37, 1672.87, 0) mm, rotated rx -180 ry 60 rz -150.43 deg; joints [-31.48, -61.018, 157.487, -1.803, -66.466, -0.235]
  MoveL 176 to (262.38, 1676.02, 0) mm, rotated rx -180 ry 60 rz -150.43 deg; joints [-31.522, -60.977, 157.134, -1.847, -66.154, -0.229]
  MoveL 177 to (266.41, 1678.5, 0) mm, rotated rx -180 ry 60 rz -150.43 deg; joints [-31.522, -60.936, 156.803, -1.851, -65.864, -0.218]
  MoveL 178 to (270.48, 1680.31, 0) mm, rotated rx -180 ry 60 rz -150.43 deg; joints [-31.482, -60.896, 156.494, -1.817, -65.595, -0.205]
  MoveL 179 to (274.58, 1681.45, 0) mm, rotated rx -180 ry 60 rz -150.43 deg; joints [-31.402, -60.856, 156.208, -1.744, -65.349, -0.188]
  MoveL 180 to (278.69, 1681.92, 0) mm, rotated rx -180 ry 60 rz -150.43 deg; joints [-31.282, -60.818, 155.945, -1.633, -65.124, -0.168]
  MoveL 181 to (282.81, 1681.7, 0) mm, rotated rx -180 ry 60 rz -150.43 deg; joints [-31.123, -60.783, 155.705, -1.483, -64.921, -0.147]
  MoveL 182 to (286.94, 1680.79, 0) mm, rotated rx -180 ry 60 rz -150.43 deg; joints [-30.925, -60.75, 155.49, -1.296, -64.739, -0.124]
  MoveL 183 to (291.06, 1679.18, 0) mm, rotated rx -180 ry 60 rz -150.43 deg; joints [-30.688, -60.719, 155.299, -1.07, -64.578, -0.099]
  MoveL 184 to (295.17, 1676.87, 0) mm, rotated rx -180 ry 60 rz -150.43 deg; joints [-30.411, -60.693, 155.132, -0.806, -64.439, -0.072]
  MoveL 185 to (299.27, 1673.86, 0) mm, rotated rx -180 ry 60 rz -150.43 deg; joints [-30.096, -60.669, 154.99, -0.504, -64.32, -0.044]
  MoveL 186 to (303.35, 1670.14, 0) mm, rotated rx -180 ry 60 rz -150.43 deg; joints [-29.742, -60.649, 154.872, -0.164, -64.222, -0.014]
  MoveL 187 to (1005.83, 1992.41, 0) mm, rotated rx 0 ry 90 rz 29.57 deg; joints [-26.974, -38.312, 110.239, 2.732, -71.946, -0.847]
  Set speed (60.0 mm/s)
  MoveL 188 to (1005.72, 1995.03, 0) mm, rotated rx 0 ry 90 rz 29.57 deg; joints [-27.071, -38.277, 110.144, 2.631, -71.885, -0.819]
  MoveL 189 to (1005.38, 1997.62, 0) mm, rotated rx 0 ry 90 rz 29.57 deg; joints [-27.171, -38.249, 110.068, 2.527, -71.835, -0.788]
  MoveL 190 to (1004.81, 2000.17, 0) mm, rotated rx 0 ry 90 rz 29.57 deg; joints [-27.274, -38.227, 110.01, 2.419, -71.798, -0.756]
  MoveL 191 to (1004.02, 2002.66, 0) mm, rotated rx 0 ry 90 rz 29.57 deg; joints [-27.378, -38.213, 109.971, 2.31, -71.772, -0.723]
  MoveL 192 to (1003.02, 2005.06, 0) mm, rotated rx 0 ry 90 rz 29.57 deg; joints [-27.483, -38.206, 109.952, 2.199, -71.759, -0.689]
  MoveL 193 to (1001.8, 2007.37, 0) mm, rotated rx 0 ry 90 rz 29.57 deg; joints [-27.589, -38.207, 109.954, 2.087, -71.759, -0.654]
  MoveL 194 to (1000.36, 2009.56, 0) mm, rotated rx 0 ry 90 rz 29.57 deg; joints [-27.695, -38.215, 109.976, 1.976, -71.771, -0.618]
  MoveL 195 to (998.72, 2011.61, 0) mm, rotated rx 0 ry 90 rz 29.57 deg; joints [-27.799, -38.231, 110.02, 1.865, -71.798, -0.583]
  MoveL 196 to (996.89, 2013.48, 0) mm, rotated rx 0 ry 90 rz 29.57 deg; joints [-27.901, -38.255, 110.085, 1.758, -71.838, -0.548]
  MoveL 197 to (994.89, 2015.15, 0) mm, rotated rx 0 ry 90 rz 29.57 deg; joints [-27.999, -38.287, 110.17, 1.654, -71.89, -0.514]
  MoveL 198 to (992.75, 2016.6, 0) mm, rotated rx 0 ry 90 rz 29.57 deg; joints [-28.092, -38.326, 110.276, 1.556, -71.956, -0.482]
  MoveL 199 to (990.48, 2017.81, 0) mm, rotated rx 0 ry 90 rz 29.57 deg; joints [-28.179, -38.372, 110.4, 1.464, -72.033, -0.452]
  MoveL 200 to (988.1, 2018.78, 0) mm, rotated rx 0 ry 90 rz 29.57 deg; joints [-28.26, -38.425, 110.543, 1.378, -72.123, -0.423]
  MoveL 201 to (985.62, 2019.49, 0) mm, rotated rx 0 ry 90 rz 29.57 deg; joints [-28.333, -38.484, 110.703, 1.3, -72.224, -0.397]
  MoveL 202 to (983.06, 2019.92, 0) mm, rotated rx 0 ry 90 rz 29.57 deg; joints [-28.399, -38.549, 110.881, 1.231, -72.335, -0.374]
  MoveL 203 to (980.43, 2020.07, 0) mm, rotated rx 0 ry 90 rz 29.57 deg; joints [-28.455, -38.621, 111.075, 1.171, -72.458, -0.353]
  MoveL 204 to (840.73, 2020.07, 0) mm, rotated rx 0 ry 90 rz 29.57 deg; joints [-31.439, -42.113, 121.178, -1.902, -79.071, 0.361]
  MoveL 205 to (840.73, 2071.02, 0) mm, rotated rx 0 ry 90 rz 29.57 deg; joints [-33.347, -41.388, 118.961, -3.866, -77.6, 0.831]
  MoveL 206 to (1043.93, 2071.02, 0) mm, rotated rx 0 ry 90 rz 29.57 deg; joints [-29.018, -35.912, 103.937, 0.597, -68.026, -0.223]
  MoveL 207 to (1043.93, 1907.58, 0) mm, rotated rx 0 ry 90 rz 29.57 deg; joints [-23.191, -38.359, 110.366, 6.706, -72.122, -2.067]
  MoveL 208 to (1015.37, 1924.76, 0) mm, rotated rx 0 ry 90 rz 29.57 deg; joints [-24.307, -38.969, 112.028, 5.502, -73.133, -1.601]
  MoveL 209 to (1005.83, 1930.45, 0) mm, rotated rx 0 ry 90 rz 29.57 deg; joints [-24.685, -39.166, 112.571, 5.098, -73.467, -1.454]
  MoveL 210 to (1000.11, 1926.67, 0) mm, rotated rx 0 ry 90 rz 29.57 deg; joints [-24.641, -39.374, 113.15, 5.134, -73.837, -1.433]
  MoveL 211 to (1001.43, 1928.6, 0) mm, rotated rx 0 ry 90 rz 29.57 deg; joints [-24.691, -39.313, 112.978, 5.085, -73.726, -1.428]
  MoveL 212 to (1002.59, 1930.63, 0) mm, rotated rx 0 ry 90 rz 29.57 deg; joints [-24.748, -39.254, 112.816, 5.029, -73.622, -1.421]
  MoveL 213 to (1003.57, 1932.75, 0) mm, rotated rx 0 ry 90 rz 29.57 deg; joints [-24.81, -39.2, 112.664, 4.966, -73.523, -1.412]
  MoveL 214 to (1004.38, 1934.94, 0) mm, rotated rx 0 ry 90 rz 29.57 deg; joints [-24.879, -39.148, 112.523, 4.897, -73.432, -1.399]
  MoveL 215 to (1005.01, 1937.19, 0) mm, rotated rx 0 ry 90 rz 29.57 deg; joints [-24.952, -39.101, 112.392, 4.822, -73.347, -1.385]
  MoveL 216 to (1005.47, 1939.49, 0) mm, rotated rx 0 ry 90 rz 29.57 deg; joints [-25.03, -39.058, 112.274, 4.743, -73.27, -1.368]
  MoveL 217 to (1005.83, 1944.16, 0) mm, rotated rx 0 ry 90 rz 29.57 deg; joints [-25.199, -38.986, 112.075, 4.57, -73.139, -1.328]
  MoveL 218 to (1005.83, 1992.41, 0) mm, rotated rx 0 ry 90 rz 29.57 deg; joints [-26.974, -38.312, 110.239, 2.732, -71.946, -0.847]
  MoveL 219 to (1041.7, 1881.48, 0) mm, rotated rx 0 ry 90 rz 29.57 deg; joints [-22.242, -38.746, 111.418, 7.674, -72.818, -2.279]
  Set speed (60.0 mm/s)
  MoveL 220 to (993.45, 1881.48, 0) mm, rotated rx 0 ry 90 rz 29.57 deg; joints [-23.016, -40.105, 115.209, 6.781, -75.203, -1.739]
  MoveL 221 to (986.57, 1882.28, 0) mm, rotated rx 0 ry 90 rz 29.57 deg; joints [-23.162, -40.282, 115.713, 6.62, -75.525, -1.662]
  MoveL 222 to (983.26, 1883.27, 0) mm, rotated rx 0 ry 90 rz 29.57 deg; joints [-23.257, -40.359, 115.935, 6.519, -75.666, -1.62]
  MoveL 223 to (980.1, 1884.64, 0) mm, rotated rx 0 ry 90 rz 29.57 deg; joints [-23.364, -40.427, 116.132, 6.404, -75.791, -1.578]
  MoveL 224 to (977.13, 1886.37, 0) mm, rotated rx 0 ry 90 rz 29.57 deg; joints [-23.483, -40.486, 116.302, 6.279, -75.898, -1.536]
  MoveL 225 to (974.39, 1888.47, 0) mm, rotated rx 0 ry 90 rz 29.57 deg; joints [-23.612, -40.534, 116.441, 6.143, -75.985, -1.493]
  MoveL 226 to (971.94, 1890.91, 0) mm, rotated rx 0 ry 90 rz 29.57 deg; joints [-23.75, -40.57, 116.547, 5.999, -76.05, -1.451]
  MoveL 227 to (969.81, 1893.7, 0) mm, rotated rx 0 ry 90 rz 29.57 deg; joints [-23.897, -40.594, 116.615, 5.847, -76.091, -1.41]
  MoveL 228 to (935.92, 1944.98, 0) mm, rotated rx 0 ry 90 rz 29.57 deg; joints [-26.518, -40.844, 117.347, 3.14, -76.522, -0.733]
  MoveL 229 to (887.38, 1944.98, 0) mm, rotated rx 0 ry 90 rz 29.57 deg; joints [-27.486, -42.017, 120.88, 2.126, -78.871, -0.41]
  MoveL 230 to (954.53, 1843.38, 0) mm, rotated rx 0 ry 90 rz 29.57 deg; joints [-22.142, -41.531, 119.393, 7.598, -77.965, -1.593]
  MoveL 231 to (1120.31, 1843.38, 0) mm, rotated rx 0 ry 90 rz 29.57 deg; joints [-19.681, -36.769, 106.149, 10.552, -69.7, -3.698]
  MoveL 232 to (1120.31, 2046.58, 0) mm, rotated rx 0 ry 90 rz 29.57 deg; joints [-26.838, -33.822, 98.682, 3.019, -64.89, -1.282]
  MoveL 233 to (1069.36, 2046.58, 0) mm, rotated rx 0 ry 90 rz 29.57 deg; joints [-27.722, -35.524, 102.947, 2.003, -67.435, -0.769]
  MoveL 234 to (1069.36, 1906.88, 0) mm, rotated rx 0 ry 90 rz 29.57 deg; joints [-22.764, -37.601, 108.336, 7.207, -70.876, -2.372]
  MoveL 235 to (1069.21, 1904.25, 0) mm, rotated rx 0 ry 90 rz 29.57 deg; joints [-22.669, -37.64, 108.438, 7.305, -70.943, -2.397]
  MoveL 236 to (1068.78, 1901.69, 0) mm, rotated rx 0 ry 90 rz 29.57 deg; joints [-22.581, -37.686, 108.56, 7.394, -71.022, -2.417]
  MoveL 237 to (1068.07, 1899.21, 0) mm, rotated rx 0 ry 90 rz 29.57 deg; joints [-22.5, -37.739, 108.702, 7.476, -71.113, -2.432]
  MoveL 238 to (1067.1, 1896.83, 0) mm, rotated rx 0 ry 90 rz 29.57 deg; joints [-22.427, -37.799, 108.861, 7.549, -71.215, -2.444]
  MoveL 239 to (1065.89, 1894.56, 0) mm, rotated rx 0 ry 90 rz 29.57 deg; joints [-22.361, -37.864, 109.036, 7.614, -71.326, -2.451]
  MoveL 240 to (1064.44, 1892.42, 0) mm, rotated rx 0 ry 90 rz 29.57 deg; joints [-22.303, -37.935, 109.225, 7.669, -71.446, -2.454]
  MoveL 241 to (1062.77, 1890.43, 0) mm, rotated rx 0 ry 90 rz 29.57 deg; joints [-22.254, -38.01, 109.427, 7.715, -71.573, -2.452]
  MoveL 242 to (1060.9, 1888.6, 0) mm, rotated rx 0 ry 90 rz 29.57 deg; joints [-22.214, -38.09, 109.639, 7.751, -71.707, -2.446]
  MoveL 243 to (1058.85, 1886.95, 0) mm, rotated rx 0 ry 90 rz 29.57 deg; joints [-22.184, -38.172, 109.86, 7.777, -71.845, -2.437]
  MoveL 244 to (1056.66, 1885.52, 0) mm, rotated rx 0 ry 90 rz 29.57 deg; joints [-22.164, -38.255, 110.084, 7.792, -71.986, -2.423]
  MoveL 245 to (1054.35, 1884.29, 0) mm, rotated rx 0 ry 90 rz 29.57 deg; joints [-22.153, -38.339, 110.31, 7.797, -72.127, -2.406]
  MoveL 246 to (1051.95, 1883.29, 0) mm, rotated rx 0 ry 90 rz 29.57 deg; joints [-22.152, -38.423, 110.537, 7.792, -72.269, -2.386]
  MoveL 247 to (1049.46, 1882.5, 0) mm, rotated rx 0 ry 90 rz 29.57 deg; joints [-22.161, -38.506, 110.763, 7.777, -72.41, -2.363]
  MoveL 248 to (1046.91, 1881.94, 0) mm, rotated rx 0 ry 90 rz 29.57 deg; joints [-22.179, -38.588, 110.986, 7.752, -72.549, -2.338]
  MoveL 249 to (1044.32, 1881.6, 0) mm, rotated rx 0 ry 90 rz 29.57 deg; joints [-22.206, -38.668, 111.205, 7.718, -72.685, -2.31]
  MoveL 250 to (1041.7, 1881.48, 0) mm, rotated rx 0 ry 90 rz 29.57 deg; joints [-22.242, -38.746, 111.418, 7.674, -72.818, -2.279]
  MoveL 251 to (892.95, 1266.65, 0) mm, rotated rx 0 ry 90 rz 29.57 deg; joints [4.332, -45.067, 131.486, 33.955, -87.029, -1.999]
  Set speed (60.0 mm/s)
  MoveL 252 to (889.54, 1266.46, 0) mm, rotated rx 0 ry 90 rz 29.57 deg; joints [4.354, -45.129, 131.741, 33.972, -87.189, -1.893]
  MoveL 253 to (886.2, 1265.88, 0) mm, rotated rx 0 ry 90 rz 29.57 deg; joints [4.396, -45.19, 131.99, 34.009, -87.346, -1.789]
  MoveL 254 to (882.94, 1264.93, 0) mm, rotated rx 0 ry 90 rz 29.57 deg; joints [4.456, -45.247, 132.228, 34.065, -87.499, -1.69]
  MoveL 255 to (879.82, 1263.61, 0) mm, rotated rx 0 ry 90 rz 29.57 deg; joints [4.535, -45.301, 132.454, 34.139, -87.644, -1.597]
  MoveL 256 to (876.88, 1266.65, 0) mm, rotated rx 0 ry 90 rz 29.57 deg; joints [4.393, -45.357, 132.693, 33.993, -87.791, -1.489]
  MoveL 257 to (825.92, 1304.75, 0) mm, rotated rx 0 ry 90 rz 29.57 deg; joints [2.58, -46.199, 136.637, 32.152, -90.371, 0.233]
  MoveL 258 to (980.11, 1304.75, 0) mm, rotated rx 0 ry 90 rz 29.57 deg; joints [2.257, -43.28, 124.947, 32.101, -82.927, -4.417]
  MoveL 259 to (1047.26, 1203.15, 0) mm, rotated rx 0 ry 90 rz 29.57 deg; joints [6.599, -41.383, 118.946, 36.821, -79.988, -7.416]
  MoveL 260 to (998.73, 1203.15, 0) mm, rotated rx 0 ry 90 rz 29.57 deg; joints [6.853, -42.637, 122.837, 36.828, -82.128, -5.856]
  MoveL 261 to (964.84, 1254.43, 0) mm, rotated rx 0 ry 90 rz 29.57 deg; joints [4.649, -43.562, 125.905, 34.46, -83.675, -4.324]
  MoveL 262 to (962.71, 1257.22, 0) mm, rotated rx 0 ry 90 rz 29.57 deg; joints [4.526, -43.615, 126.089, 34.328, -83.773, -4.236]
  MoveL 263 to (960.25, 1259.66, 0) mm, rotated rx 0 ry 90 rz 29.57 deg; joints [4.42, -43.675, 126.294, 34.213, -83.886, -4.142]
  MoveL 264 to (957.52, 1261.76, 0) mm, rotated rx 0 ry 90 rz 29.57 deg; joints [4.331, -43.74, 126.52, 34.115, -84.012, -4.042]
  MoveL 265 to (954.55, 1263.49, 0) mm, rotated rx 0 ry 90 rz 29.57 deg; joints [4.26, -43.808, 126.76, 34.033, -84.15, -3.938]
  MoveL 266 to (951.38, 1264.86, 0) mm, rotated rx 0 ry 90 rz 29.57 deg; joints [4.206, -43.88, 127.013, 33.969, -84.296, -3.831]
  MoveL 267 to (948.07, 1265.85, 0) mm, rotated rx 0 ry 90 rz 29.57 deg; joints [4.171, -43.954, 127.275, 33.923, -84.45, -3.722]
  MoveL 268 to (941.19, 1266.65, 0) mm, rotated rx 0 ry 90 rz 29.57 deg; joints [4.157, -44.103, 127.81, 33.888, -84.769, -3.504]
  MoveL 269 to (892.95, 1266.65, 0) mm, rotated rx 0 ry 90 rz 29.57 deg; joints [4.332, -45.067, 131.486, 33.955, -87.029, -1.999]
  MoveL 270 to (1053.1, 1149.78, 0) mm, rotated rx 0 ry 90 rz 29.57 deg; joints [8.873, -41.026, 117.881, 39.188, -79.74, -8.262]
  Set speed (60.0 mm/s)
  MoveL 271 to (898.67, 1149.78, 0) mm, rotated rx 0 ry 90 rz 29.57 deg; joints [10.043, -44.676, 129.943, 39.711, -86.355, -3.022]
  MoveL 272 to (894.63, 1149.99, 0) mm, rotated rx 0 ry 90 rz 29.57 deg; joints [10.068, -44.755, 130.249, 39.726, -86.531, -2.879]
  MoveL 273 to (890.72, 1150.63, 0) mm, rotated rx 0 ry 90 rz 29.57 deg; joints [10.071, -44.833, 130.55, 39.721, -86.704, -2.735]
  MoveL 274 to (886.94, 1151.67, 0) mm, rotated rx 0 ry 90 rz 29.57 deg; joints [10.052, -44.908, 130.847, 39.695, -86.873, -2.592]
  MoveL 275 to (883.33, 1153.13, 0) mm, rotated rx 0 ry 90 rz 29.57 deg; joints [10.012, -44.98, 131.135, 39.647, -87.038, -2.452]
  MoveL 276 to (879.91, 1154.97, 0) mm, rotated rx 0 ry 90 rz 29.57 deg; joints [9.951, -45.049, 131.415, 39.579, -87.197, -2.315]
  MoveL 277 to (876.69, 1157.21, 0) mm, rotated rx 0 ry 90 rz 29.57 deg; joints [9.869, -45.115, 131.683, 39.491, -87.35, -2.182]
  MoveL 278 to (873.71, 1159.83, 0) mm, rotated rx 0 ry 90 rz 29.57 deg; joints [9.765, -45.177, 131.938, 39.381, -87.495, -2.054]
  MoveL 279 to (870.99, 1162.83, 0) mm, rotated rx 0 ry 90 rz 29.57 deg; joints [9.639, -45.235, 132.178, 39.251, -87.632, -1.933]
  MoveL 280 to (868.67, 1166, 0) mm, rotated rx 0 ry 90 rz 29.57 deg; joints [9.501, -45.285, 132.39, 39.108, -87.753, -1.826]
  MoveL 281 to (866.69, 1169.36, 0) mm, rotated rx 0 ry 90 rz 29.57 deg; joints [9.349, -45.33, 132.578, 38.953, -87.859, -1.73]
  MoveL 282 to (865.04, 1172.89, 0) mm, rotated rx 0 ry 90 rz 29.57 deg; joints [9.187, -45.369, 132.743, 38.787, -87.953, -1.645]
  MoveL 283 to (863.72, 1176.55, 0) mm, rotated rx 0 ry 90 rz 29.57 deg; joints [9.014, -45.402, 132.884, 38.612, -88.032, -1.571]
  MoveL 284 to (862.71, 1180.31, 0) mm, rotated rx 0 ry 90 rz 29.57 deg; joints [8.833, -45.429, 133.003, 38.43, -88.099, -1.508]
  MoveL 285 to (862, 1184.14, 0) mm, rotated rx 0 ry 90 rz 29.57 deg; joints [8.646, -45.451, 133.099, 38.241, -88.152, -1.456]
  MoveL 286 to (861.58, 1188.01, 0) mm, rotated rx 0 ry 90 rz 29.57 deg; joints [8.453, -45.468, 133.173, 38.047, -88.192, -1.415]
  MoveL 287 to (861.44, 1191.9, 0) mm, rotated rx 0 ry 90 rz 29.57 deg; joints [8.258, -45.48, 133.225, 37.851, -88.219, -1.384]
  MoveL 288 to (861.44, 1246.06, 0) mm, rotated rx 0 ry 90 rz 29.57 deg; joints [5.507, -45.59, 133.71, 35.093, -88.461, -1.081]
  MoveL 289 to (823.34, 1246.06, 0) mm, rotated rx 0 ry 90 rz 29.57 deg; joints [5.701, -46.175, 136.515, 35.273, -90.277, 0.196]
  MoveL 290 to (823.34, 1108.29, 0) mm, rotated rx 0 ry 90 rz 29.57 deg; joints [12.854, -45.844, 134.874, 42.43, -89.284, -0.654]
  MoveL 291 to (1061.99, 1108.29, 0) mm, rotated rx 0 ry 90 rz 29.57 deg; joints [10.574, -40.58, 116.575, 41, -79.34, -9.135]
  MoveL 292 to (1059.69, 1118.65, 0) mm, rotated rx 0 ry 90 rz 29.57 deg; joints [10.154, -40.698, 116.918, 40.55, -79.444, -8.908]
  MoveL 293 to (1053.1, 1149.78, 0) mm, rotated rx 0 ry 90 rz 29.57 deg; joints [8.873, -41.026, 117.881, 39.188, -79.74, -8.262]
  MoveL 294 to (824.97, 1409.86, 0) mm, rotated rx 0 ry 90 rz 29.57 deg; joints [-3.016, -46.206, 136.677, 26.557, -90.421, 0.21]
  Set speed (60.0 mm/s)
  MoveL 295 to (822.36, 1409.74, 0) mm, rotated rx 0 ry 90 rz 29.57 deg; joints [-3.017, -46.243, 136.869, 26.556, -90.56, 0.28]
  MoveL 296 to (819.76, 1409.4, 0) mm, rotated rx 0 ry 90 rz 29.57 deg; joints [-3.006, -46.278, 137.06, 26.568, -90.699, 0.349]
  MoveL 297 to (817.21, 1408.83, 0) mm, rotated rx 0 ry 90 rz 29.57 deg; joints [-2.983, -46.313, 137.248, 26.592, -90.836, 0.418]
  MoveL 298 to (814.73, 1408.05, 0) mm, rotated rx 0 ry 90 rz 29.57 deg; joints [-2.947, -46.347, 137.432, 26.628, -90.971, 0.487]
  MoveL 299 to (812.32, 1407.04, 0) mm, rotated rx 0 ry 90 rz 29.57 deg; joints [-2.9, -46.379, 137.611, 26.677, -91.101, 0.553]
  MoveL 300 to (810.02, 1405.82, 0) mm, rotated rx 0 ry 90 rz 29.57 deg; joints [-2.841, -46.409, 137.784, 26.738, -91.227, 0.618]
  MoveL 301 to (807.83, 1404.39, 0) mm, rotated rx 0 ry 90 rz 29.57 deg; joints [-2.769, -46.438, 137.948, 26.811, -91.347, 0.681]
  MoveL 302 to (805.78, 1402.74, 0) mm, rotated rx 0 ry 90 rz 29.57 deg; joints [-2.685, -46.465, 138.102, 26.896, -91.461, 0.741]
  MoveL 303 to (803.9, 1400.91, 0) mm, rotated rx 0 ry 90 rz 29.57 deg; joints [-2.59, -46.489, 138.245, 26.992, -91.564, 0.797]
  MoveL 304 to (802.24, 1398.91, 0) mm, rotated rx 0 ry 90 rz 29.57 deg; joints [-2.486, -46.511, 138.372, 27.098, -91.657, 0.848]
  MoveL 305 to (800.79, 1396.77, 0) mm, rotated rx 0 ry 90 rz 29.57 deg; joints [-2.373, -46.529, 138.484, 27.212, -91.738, 0.894]
  MoveL 306 to (799.57, 1394.51, 0) mm, rotated rx 0 ry 90 rz 29.57 deg; joints [-2.252, -46.545, 138.578, 27.334, -91.806, 0.933]
  MoveL 307 to (798.61, 1392.12, 0) mm, rotated rx 0 ry 90 rz 29.57 deg; joints [-2.124, -46.558, 138.655, 27.463, -91.861, 0.967]
  MoveL 308 to (797.9, 1389.64, 0) mm, rotated rx 0 ry 90 rz 29.57 deg; joints [-1.99, -46.567, 138.713, 27.598, -91.902, 0.994]
  MoveL 309 to (797.46, 1387.08, 0) mm, rotated rx 0 ry 90 rz 29.57 deg; joints [-1.851, -46.573, 138.75, 27.737, -91.927, 1.013]
  MoveL 310 to (797.32, 1384.46, 0) mm, rotated rx 0 ry 90 rz 29.57 deg; joints [-1.708, -46.576, 138.767, 27.881, -91.937, 1.024]
  MoveL 311 to (797.32, 1108.32, 0) mm, rotated rx 0 ry 90 rz 29.57 deg; joints [13.161, -46.219, 136.743, 42.734, -90.385, 0.355]
  MoveL 312 to (746.36, 1146.42, 0) mm, rotated rx 0 ry 90 rz 29.57 deg; joints [11.725, -46.895, 140.939, 41.368, -93.037, 2.672]
  MoveL 313 to (746.36, 1447.96, 0) mm, rotated rx 0 ry 90 rz 29.57 deg; joints [-5.431, -47.038, 142.132, 24.225, -94.648, 2.088]
  MoveL 314 to (912.14, 1447.96, 0) mm, rotated rx 0 ry 90 rz 29.57 deg; joints [-4.66, -44.687, 129.985, 24.986, -85.736, -1.984]
  MoveL 315 to (979.29, 1346.36, 0) mm, rotated rx 0 ry 90 rz 29.57 deg; joints [0.32, -43.321, 125.085, 30.149, -82.866, -4.126]
  MoveL 316 to (930.76, 1346.36, 0) mm, rotated rx 0 ry 90 rz 29.57 deg; joints [0.333, -44.389, 128.854, 30.021, -85.204, -2.766]
  MoveL 317 to (896.87, 1397.63, 0) mm, rotated rx 0 ry 90 rz 29.57 deg; joints [-2.217, -45.039, 131.372, 27.402, -86.744, -1.687]
  MoveL 318 to (894.74, 1400.42, 0) mm, rotated rx 0 ry 90 rz 29.57 deg; joints [-2.361, -45.076, 131.525, 27.255, -86.842, -1.626]
  MoveL 319 to (892.28, 1402.87, 0) mm, rotated rx 0 ry 90 rz 29.57 deg; joints [-2.488, -45.12, 131.702, 27.124, -86.957, -1.558]
  MoveL 320 to (889.55, 1404.96, 0) mm, rotated rx 0 ry 90 rz 29.57 deg; joints [-2.6, -45.168, 131.901, 27.01, -87.089, -1.483]
  MoveL 321 to (886.57, 1406.7, 0) mm, rotated rx 0 ry 90 rz 29.57 deg; joints [-2.694, -45.221, 132.119, 26.912, -87.233, -1.403]
  MoveL 322 to (883.41, 1408.07, 0) mm, rotated rx 0 ry 90 rz 29.57 deg; joints [-2.77, -45.276, 132.352, 26.832, -87.39, -1.32]
  MoveL 323 to (880.1, 1409.05, 0) mm, rotated rx 0 ry 90 rz 29.57 deg; joints [-2.828, -45.334, 132.596, 26.77, -87.555, -1.233]
  MoveL 324 to (873.22, 1409.86, 0) mm, rotated rx 0 ry 90 rz 29.57 deg; joints [-2.886, -45.453, 133.108, 26.705, -87.905, -1.054]
  MoveL 325 to (824.97, 1409.86, 0) mm, rotated rx 0 ry 90 rz 29.57 deg; joints [-3.016, -46.206, 136.677, 26.557, -90.421, 0.21]
  MoveL 326 to (667.84, 1086.24, 0) mm, rotated rx 0 ry 90 rz 29.57 deg; joints [16.218, -47.292, 145.296, 46.07, -95.572, 5.755]
  Set speed (60.0 mm/s)
  MoveL 327 to (664.42, 1088.09, 0) mm, rotated rx 0 ry 90 rz 29.57 deg; joints [16.169, -47.304, 145.561, 46.039, -95.752, 5.933]
  MoveL 328 to (661.2, 1090.32, 0) mm, rotated rx 0 ry 90 rz 29.57 deg; joints [16.093, -47.315, 145.819, 45.981, -95.932, 6.105]
  MoveL 329 to (658.22, 1092.94, 0) mm, rotated rx 0 ry 90 rz 29.57 deg; joints [15.99, -47.323, 146.068, 45.897, -96.11, 6.268]
  MoveL 330 to (655.5, 1095.94, 0) mm, rotated rx 0 ry 90 rz 29.57 deg; joints [15.861, -47.33, 146.307, 45.785, -96.286, 6.421]
  MoveL 331 to (653.18, 1099.11, 0) mm, rotated rx 0 ry 90 rz 29.57 deg; joints [15.713, -47.335, 146.521, 45.655, -96.449, 6.555]
  MoveL 332 to (651.2, 1102.47, 0) mm, rotated rx 0 ry 90 rz 29.57 deg; joints [15.548, -47.339, 146.715, 45.505, -96.602, 6.674]
  MoveL 333 to (649.55, 1106, 0) mm, rotated rx 0 ry 90 rz 29.57 deg; joints [15.366, -47.341, 146.89, 45.338, -96.744, 6.776]
  MoveL 334 to (648.23, 1109.66, 0) mm, rotated rx 0 ry 90 rz 29.57 deg; joints [15.171, -47.343, 147.044, 45.155, -96.874, 6.862]
  MoveL 335 to (647.22, 1113.42, 0) mm, rotated rx 0 ry 90 rz 29.57 deg; joints [14.963, -47.344, 147.179, 44.959, -96.994, 6.933]
  MoveL 336 to (646.51, 1117.25, 0) mm, rotated rx 0 ry 90 rz 29.57 deg; joints [14.746, -47.344, 147.294, 44.752, -97.101, 6.987]
  MoveL 337 to (646.09, 1121.13, 0) mm, rotated rx 0 ry 90 rz 29.57 deg; joints [14.52, -47.344, 147.389, 44.534, -97.197, 7.027]
  MoveL 338 to (645.95, 1125.01, 0) mm, rotated rx 0 ry 90 rz 29.57 deg; joints [14.289, -47.344, 147.465, 44.31, -97.279, 7.051]
  MoveL 339 to (645.95, 1228.44, 0) mm, rotated rx 0 ry 90 rz 29.57 deg; joints [7.929, -47.316, 148.831, 38.064, -99.112, 7.07]
  MoveL 340 to (607.85, 1228.44, 0) mm, rotated rx 0 ry 90 rz 29.57 deg; joints [8.276, -47.118, 151.381, 38.72, -101.218, 8.865]
  MoveL 341 to (607.85, 1041.4, 0) mm, rotated rx 0 ry 90 rz 29.57 deg; joints [19.975, -47.334, 148.274, 50.064, -97.073, 8.367]
  MoveL 342 to (1071.45, 1041.4, 0) mm, rotated rx 0 ry 90 rz 29.57 deg; joints [13.277, -39.906, 114.642, 43.875, -78.871, -10.513]
  MoveL 343 to (1066.6, 1051.72, 0) mm, rotated rx 0 ry 90 rz 29.57 deg; joints [12.898, -40.115, 115.236, 43.444, -79.082, -10.17]
  MoveL 344 to (1052.59, 1082.89, 0) mm, rotated rx 0 ry 90 rz 29.57 deg; joints [11.724, -40.703, 116.934, 42.125, -79.699, -9.187]
  MoveL 345 to (683.18, 1082.89, 0) mm, rotated rx 0 ry 90 rz 29.57 deg; joints [16.155, -47.227, 144.201, 45.939, -94.863, 5.006]
  MoveL 346 to (679.15, 1083.11, 0) mm, rotated rx 0 ry 90 rz 29.57 deg; joints [16.209, -47.245, 144.477, 46.009, -95.036, 5.196]
  MoveL 347 to (675.23, 1083.74, 0) mm, rotated rx 0 ry 90 rz 29.57 deg; joints [16.238, -47.263, 144.752, 46.055, -95.213, 5.385]
  MoveL 348 to (671.45, 1084.79, 0) mm, rotated rx 0 ry 90 rz 29.57 deg; joints [16.241, -47.278, 145.026, 46.075, -95.392, 5.572]
  MoveL 349 to (667.84, 1086.24, 0) mm, rotated rx 0 ry 90 rz 29.57 deg; joints [16.218, -47.292, 145.296, 46.07, -95.572, 5.755]
  MoveL 350 to (819.97, 1615.51, 0) mm, rotated rx 0 ry 90 rz 29.57 deg; joints [-13.773, -45.833, 134.821, 15.801, -89.027, -0.275]
  Set speed (60.0 mm/s)
  MoveL 351 to (815.87, 1618.52, 0) mm, rotated rx 0 ry 90 rz 29.57 deg; joints [-13.977, -45.883, 135.062, 15.597, -89.209, -0.221]
  MoveL 352 to (811.76, 1620.83, 0) mm, rotated rx 0 ry 90 rz 29.57 deg; joints [-14.146, -45.936, 135.316, 15.427, -89.402, -0.165]
  MoveL 353 to (807.64, 1622.44, 0) mm, rotated rx 0 ry 90 rz 29.57 deg; joints [-14.28, -45.991, 135.582, 15.292, -89.605, -0.108]
  MoveL 354 to (803.51, 1623.35, 0) mm, rotated rx 0 ry 90 rz 29.57 deg; joints [-14.38, -46.047, 135.86, 15.191, -89.819, -0.049]
  MoveL 355 to (799.39, 1623.57, 0) mm, rotated rx 0 ry 90 rz 29.57 deg; joints [-14.446, -46.104, 136.149, 15.126, -90.044, 0.012]
  MoveL 356 to (795.28, 1623.11, 0) mm, rotated rx 0 ry 90 rz 29.57 deg; joints [-14.476, -46.163, 136.45, 15.095, -90.277, 0.075]
  MoveL 357 to (791.18, 1621.96, 0) mm, rotated rx 0 ry 90 rz 29.57 deg; joints [-14.472, -46.223, 136.762, 15.1, -90.521, 0.141]
  MoveL 358 to (787.11, 1620.15, 0) mm, rotated rx 0 ry 90 rz 29.57 deg; joints [-14.433, -46.283, 137.084, 15.14, -90.773, 0.209]
  MoveL 359 to (783.08, 1617.67, 0) mm, rotated rx 0 ry 90 rz 29.57 deg; joints [-14.357, -46.343, 137.414, 15.217, -91.033, 0.281]
  MoveL 360 to (779.07, 1614.52, 0) mm, rotated rx 0 ry 90 rz 29.57 deg; joints [-14.247, -46.404, 137.754, 15.329, -91.302, 0.357]
  MoveL 361 to (775.12, 1610.72, 0) mm, rotated rx 0 ry 90 rz 29.57 deg; joints [-14.1, -46.464, 138.101, 15.478, -91.577, 0.437]
  MoveL 362 to (767.37, 1601.17, 0) mm, rotated rx 0 ry 90 rz 29.57 deg; joints [-13.696, -46.583, 138.813, 15.887, -92.144, 0.61]
  MoveL 363 to (761.62, 1592.15, 0) mm, rotated rx 0 ry 90 rz 29.57 deg; joints [-13.288, -46.671, 139.369, 16.301, -92.589, 0.757]
  MoveL 364 to (756.45, 1582.48, 0) mm, rotated rx 0 ry 90 rz 29.57 deg; joints [-12.832, -46.749, 139.889, 16.763, -93.006, 0.905]
  MoveL 365 to (747.84, 1562.64, 0) mm, rotated rx 0 ry 90 rz 29.57 deg; joints [-11.852, -46.876, 140.797, 17.759, -93.735, 1.195]
  MoveL 366 to (740.38, 1540.88, 0) mm, rotated rx 0 ry 90 rz 29.57 deg; joints [-10.728, -46.98, 141.624, 18.901, -94.395, 1.503]
  MoveL 367 to (728.8, 1495.08, 0) mm, rotated rx 0 ry 90 rz 29.57 deg; joints [-8.246, -47.124, 142.97, 21.427, -95.445, 2.133]
  MoveL 368 to (721.23, 1451.76, 0) mm, rotated rx 0 ry 90 rz 29.57 deg; joints [-5.793, -47.202, 143.873, 23.923, -96.102, 2.7]
  MoveL 369 to (714.36, 1388.82, 0) mm, rotated rx 0 ry 90 rz 29.57 deg; joints [-2.114, -47.257, 144.658, 27.654, -96.564, 3.428]
  MoveL 370 to (711.2, 1304.56, 0) mm, rotated rx 0 ry 90 rz 29.57 deg; joints [2.898, -47.268, 144.839, 32.697, -96.382, 4.082]
  MoveL 371 to (711.2, 1115.64, 0) mm, rotated rx 0 ry 90 rz 29.57 deg; joints [13.883, -47.117, 142.892, 43.6, -94.189, 3.98]
  MoveL 372 to (673.1, 1115.64, 0) mm, rotated rx 0 ry 90 rz 29.57 deg; joints [14.433, -47.301, 145.484, 44.297, -95.876, 5.705]
  MoveL 373 to (673.1, 1968.88, 0) mm, rotated rx 0 ry 90 rz 29.57 deg; joints [-33.7, -45.706, 134.234, -4.13, -88.531, 0.106]
  MoveL 374 to (1130.3, 1335.87, 0) mm, rotated rx 0 ry 90 rz 29.57 deg; joints [0.72, -39.219, 112.718, 31.352, -75.803, -8.498]
  MoveL 375 to (1130.3, 1042.48, 0) mm, rotated rx 0 ry 90 rz 29.57 deg; joints [12.687, -38.127, 109.741, 43.756, -76.499, -12.6]
  MoveL 376 to (1092.2, 1121.07, 0) mm, rotated rx 0 ry 90 rz 29.57 deg; joints [9.813, -39.775, 114.272, 40.429, -78.078, -9.982]
  MoveL 377 to (1085.99, 1117.44, 0) mm, rotated rx 0 ry 90 rz 29.57 deg; joints [10.008, -39.939, 114.735, 40.585, -78.339, -9.823]
  MoveL 378 to (1081.58, 1154.26, 0) mm, rotated rx 0 ry 90 rz 29.57 deg; joints [8.498, -40.242, 115.599, 38.991, -78.521, -9.152]
  MoveL 379 to (1068.65, 1225.33, 0) mm, rotated rx 0 ry 90 rz 29.57 deg; joints [5.539, -40.859, 117.39, 35.866, -79.016, -7.844]
  MoveL 380 to (1058.35, 1263.64, 0) mm, rotated rx 0 ry 90 rz 29.57 deg; joints [3.917, -41.233, 118.495, 34.149, -79.404, -7.11]
  MoveL 381 to (1051.94, 1282.64, 0) mm, rotated rx 0 ry 90 rz 29.57 deg; joints [3.103, -41.439, 119.114, 33.285, -79.649, -6.727]
  MoveL 382 to (1044.63, 1300.77, 0) mm, rotated rx 0 ry 90 rz 29.57 deg; joints [2.32, -41.659, 119.779, 32.451, -79.934, -6.341]
  MoveL 383 to (1027.17, 1332.11, 0) mm, rotated rx 0 ry 90 rz 29.57 deg; joints [0.947, -42.141, 121.264, 30.975, -80.645, -5.573]
  MoveL 384 to (832.1, 1602.19, 0) mm, rotated rx 0 ry 90 rz 29.57 deg; joints [-12.957, -45.693, 134.173, 16.621, -88.544, -0.435]
  MoveL 385 to (824.05, 1611.79, 0) mm, rotated rx 0 ry 90 rz 29.57 deg; joints [-13.535, -45.784, 134.592, 16.04, -88.855, -0.329]
  MoveL 386 to (819.97, 1615.51, 0) mm, rotated rx 0 ry 90 rz 29.57 deg; joints [-13.773, -45.833, 134.821, 15.801, -89.027, -0.275]
  MoveL 387 to (1051.03, 1672.5, 0) mm, rotated rx 0 ry 90 rz 29.57 deg; joints [-13.788, -40.437, 116.161, 16.261, -76.273, -3.959]
  Set speed (60.0 mm/s)
  MoveL 388 to (1042.85, 1679.23, 0) mm, rotated rx 0 ry 90 rz 29.57 deg; joints [-14.152, -40.618, 116.686, 15.863, -76.579, -3.774]
  MoveL 389 to (1034.8, 1688.83, 0) mm, rotated rx 0 ry 90 rz 29.57 deg; joints [-14.639, -40.772, 117.135, 15.346, -76.832, -3.577]
  MoveL 390 to (839.73, 1958.92, 0) mm, rotated rx 0 ry 90 rz 29.57 deg; joints [-29.065, -42.907, 123.71, 0.513, -80.804, -0.082]
  MoveL 391 to (822.27, 1990.25, 0) mm, rotated rx 0 ry 90 rz 29.57 deg; joints [-30.713, -42.895, 123.672, -1.157, -80.779, 0.185]
  MoveL 392 to (814.96, 2008.38, 0) mm, rotated rx 0 ry 90 rz 29.57 deg; joints [-31.599, -42.819, 123.424, -2.054, -80.611, 0.335]
  MoveL 393 to (808.55, 2027.39, 0) mm, rotated rx 0 ry 90 rz 29.57 deg; joints [-32.491, -42.705, 123.054, -2.961, -80.362, 0.496]
  MoveL 394 to (798.26, 2065.69, 0) mm, rotated rx 0 ry 90 rz 29.57 deg; joints [-34.202, -42.394, 122.059, -4.706, -79.7, 0.843]
  MoveL 395 to (787.07, 2124.74, 0) mm, rotated rx 0 ry 90 rz 29.57 deg; joints [-36.646, -41.742, 120.034, -7.223, -78.382, 1.462]
  MoveL 396 to (778.57, 2199.46, 0) mm, rotated rx 0 ry 90 rz 29.57 deg; joints [-39.444, -40.658, 116.802, -10.162, -76.353, 2.422]
  MoveL 397 to (774.7, 2299.07, 0) mm, rotated rx 0 ry 90 rz 29.57 deg; joints [-42.707, -38.78, 111.509, -13.733, -73.195, 4.041]
  MoveL 398 to (774.7, 2323, 0) mm, rotated rx 0 ry 90 rz 29.57 deg; joints [-43.421, -38.258, 110.091, -14.546, -72.379, 4.491]
  MoveL 399 to (736.6, 2401.6, 0) mm, rotated rx 0 ry 90 rz 29.57 deg; joints [-46.737, -37.307, 107.558, -18.17, -71.165, 6.048]
  MoveL 400 to (736.6, 1955.16, 0) mm, rotated rx 0 ry 90 rz 29.57 deg; joints [-31.386, -44.888, 130.767, -1.82, -85.881, 0.131]
  MoveL 401 to (1193.8, 1322.14, 0) mm, rotated rx 0 ry 90 rz 29.57 deg; joints [1.233, -37.153, 107.153, 32.395, -72.916, -10.558]
  MoveL 402 to (1193.8, 2290.27, 0) mm, rotated rx 0 ry 90 rz 29.57 deg; joints [-32.983, -25.482, 79.018, -4.239, -53.611, 2.518]
  MoveL 403 to (1155.7, 2290.27, 0) mm, rotated rx 0 ry 90 rz 29.57 deg; joints [-33.687, -27.101, 82.716, -4.982, -55.716, 2.811]
  MoveL 404 to (1155.7, 1986.46, 0) mm, rotated rx 0 ry 90 rz 29.57 deg; joints [-24.25, -33.588, 98.103, 5.891, -64.634, -2.531]
  MoveL 405 to (1152.54, 1902.21, 0) mm, rotated rx 0 ry 90 rz 29.57 deg; joints [-21.376, -34.946, 101.486, 8.923, -66.793, -3.54]
  MoveL 406 to (1148.44, 1860.23, 0) mm, rotated rx 0 ry 90 rz 29.57 deg; joints [-19.928, -35.631, 103.218, 10.415, -67.921, -3.952]
  MoveL 407 to (1142.38, 1818.5, 0) mm, rotated rx 0 ry 90 rz 29.57 deg; joints [-18.477, -36.325, 104.999, 11.888, -69.091, -4.296]
  MoveL 408 to (1132.84, 1772.91, 0) mm, rotated rx 0 ry 90 rz 29.57 deg; joints [-16.882, -37.119, 107.064, 13.479, -70.455, -4.585]
  MoveL 409 to (1126.52, 1750.15, 0) mm, rotated rx 0 ry 90 rz 29.57 deg; joints [-16.084, -37.542, 108.178, 14.264, -71.191, -4.686]
  MoveL 410 to (1119.06, 1728.39, 0) mm, rotated rx 0 ry 90 rz 29.57 deg; joints [-15.324, -37.974, 109.33, 15.002, -71.949, -4.747]
  MoveL 411 to (1110.45, 1708.54, 0) mm, rotated rx 0 ry 90 rz 29.57 deg; joints [-14.637, -38.411, 110.505, 15.659, -72.719, -4.76]
  MoveL 412 to (1105.28, 1698.87, 0) mm, rotated rx 0 ry 90 rz 29.57 deg; joints [-14.307, -38.648, 111.148, 15.968, -73.137, -4.745]
  MoveL 413 to (1099.53, 1689.86, 0) mm, rotated rx 0 ry 90 rz 29.57 deg; joints [-14.006, -38.893, 111.82, 16.246, -73.571, -4.712]
  MoveL 414 to (1091.78, 1680.3, 0) mm, rotated rx 0 ry 90 rz 29.57 deg; joints [-13.699, -39.199, 112.662, 16.521, -74.111, -4.643]
  MoveL 415 to (1083.83, 1673.36, 0) mm, rotated rx 0 ry 90 rz 29.57 deg; joints [-13.496, -39.486, 113.46, 16.69, -74.617, -4.547]
  MoveL 416 to (1079.79, 1670.87, 0) mm, rotated rx 0 ry 90 rz 29.57 deg; joints [-13.434, -39.622, 113.843, 16.735, -74.857, -4.491]
  MoveL 417 to (1075.72, 1669.06, 0) mm, rotated rx 0 ry 90 rz 29.57 deg; joints [-13.4, -39.754, 114.214, 16.752, -75.089, -4.429]
  MoveL 418 to (1071.62, 1667.92, 0) mm, rotated rx 0 ry 90 rz 29.57 deg; joints [-13.393, -39.881, 114.572, 16.741, -75.311, -4.362]
  MoveL 419 to (1067.51, 1667.46, 0) mm, rotated rx 0 ry 90 rz 29.57 deg; joints [-13.414, -40.003, 114.918, 16.702, -75.524, -4.289]
  MoveL 420 to (1063.39, 1667.68, 0) mm, rotated rx 0 ry 90 rz 29.57 deg; joints [-13.464, -40.12, 115.251, 16.635, -75.727, -4.213]
  MoveL 421 to (1059.27, 1668.59, 0) mm, rotated rx 0 ry 90 rz 29.57 deg; joints [-13.542, -40.231, 115.569, 16.54, -75.92, -4.132]
  MoveL 422 to (1055.14, 1670.19, 0) mm, rotated rx 0 ry 90 rz 29.57 deg; joints [-13.65, -40.337, 115.873, 16.415, -76.102, -4.047]
  MoveL 423 to (1051.03, 1672.5, 0) mm, rotated rx 0 ry 90 rz 29.57 deg; joints [-13.788, -40.437, 116.161, 16.261, -76.273, -3.959]
  MoveL 424 to (152.4, 2122.08, 0) mm, rotated rx 0 ry 90 rz 29.57 deg; joints [-62.371, -47.125, 151.321, -33.613, -101.896, -7.802]
  Set speed (60.0 mm/s)
  MoveL 425 to (242.26, 2181.47, 0) mm, rotated rx 0 ry 90 rz 29.57 deg; joints [-59.273, -47.264, 144.767, -29.914, -96.513, -3.734]
  MoveL 426 to (245.1, 2183.49, 0) mm, rotated rx 0 ry 90 rz 29.57 deg; joints [-59.189, -47.25, 144.544, -29.818, -96.337, -3.62]
  MoveL 427 to (247.78, 2185.69, 0) mm, rotated rx 0 ry 90 rz 29.57 deg; joints [-59.12, -47.235, 144.315, -29.737, -96.156, -3.505]
  MoveL 428 to (250.31, 2188.06, 0) mm, rotated rx 0 ry 90 rz 29.57 deg; joints [-59.064, -47.218, 144.082, -29.669, -95.971, -3.391]
  MoveL 429 to (252.67, 2190.59, 0) mm, rotated rx 0 ry 90 rz 29.57 deg; joints [-59.021, -47.2, 143.844, -29.615, -95.782, -3.278]
  MoveL 430 to (254.87, 2193.27, 0) mm, rotated rx 0 ry 90 rz 29.57 deg; joints [-58.992, -47.18, 143.603, -29.575, -95.591, -3.165]
  MoveL 431 to (256.89, 2196.08, 0) mm, rotated rx 0 ry 90 rz 29.57 deg; joints [-58.975, -47.16, 143.359, -29.548, -95.399, -3.053]
  MoveL 432 to (258.73, 2199.02, 0) mm, rotated rx 0 ry 90 rz 29.57 deg; joints [-58.971, -47.138, 143.114, -29.533, -95.205, -2.942]
  MoveL 433 to (260.4, 2202.07, 0) mm, rotated rx 0 ry 90 rz 29.57 deg; joints [-58.98, -47.114, 142.869, -29.532, -95.011, -2.833]
  MoveL 434 to (261.87, 2205.21, 0) mm, rotated rx 0 ry 90 rz 29.57 deg; joints [-59, -47.09, 142.625, -29.544, -94.819, -2.726]
  MoveL 435 to (263.14, 2208.43, 0) mm, rotated rx 0 ry 90 rz 29.57 deg; joints [-59.033, -47.065, 142.383, -29.567, -94.629, -2.621]
  MoveL 436 to (264.23, 2211.71, 0) mm, rotated rx 0 ry 90 rz 29.57 deg; joints [-59.076, -47.039, 142.144, -29.602, -94.441, -2.519]
  MoveL 437 to (265.11, 2215.05, 0) mm, rotated rx 0 ry 90 rz 29.57 deg; joints [-59.131, -47.013, 141.908, -29.649, -94.257, -2.419]
  MoveL 438 to (265.81, 2218.43, 0) mm, rotated rx 0 ry 90 rz 29.57 deg; joints [-59.196, -46.986, 141.676, -29.707, -94.076, -2.322]
  MoveL 439 to (266.3, 2221.85, 0) mm, rotated rx 0 ry 90 rz 29.57 deg; joints [-59.271, -46.959, 141.448, -29.775, -93.899, -2.228]
  MoveL 440 to (266.6, 2225.3, 0) mm, rotated rx 0 ry 90 rz 29.57 deg; joints [-59.356, -46.931, 141.226, -29.854, -93.727, -2.136]
  MoveL 441 to (266.7, 2228.76, 0) mm, rotated rx 0 ry 90 rz 29.57 deg; joints [-59.45, -46.904, 141.01, -29.943, -93.559, -2.048]
  MoveL 442 to (266.7, 2374.4, 0) mm, rotated rx 0 ry 90 rz 29.57 deg; joints [-63.159, -45.1, 131.621, -33.636, -87.103, 1.926]
  MoveL 443 to (304.8, 2374.4, 0) mm, rotated rx 0 ry 90 rz 29.57 deg; joints [-61.483, -44.763, 130.28, -31.99, -86.195, 2.374]
  MoveL 444 to (304.8, 2174.27, 0) mm, rotated rx 0 ry 90 rz 29.57 deg; joints [-55.95, -47.111, 142.838, -26.493, -95.129, -2.551]
  MoveL 445 to (152.4, 2073.55, 0) mm, rotated rx 0 ry 90 rz 29.57 deg; joints [-60.808, -46.643, 154.153, -32.454, -104.907, -9.291]
  MoveL 446 to (152.4, 2122.08, 0) mm, rotated rx 0 ry 90 rz 29.57 deg; joints [-62.371, -47.125, 151.321, -33.613, -101.896, -7.802]
  MoveL 447 to (1113.37, 952.5, 0) mm, rotated rx 0 ry 90 rz 29.57 deg; joints [16.378, -37.925, 109.198, 47.505, -77.101, -13.694]
  Set speed (60.0 mm/s)
  MoveL 448 to (88.9, 952.5, 0) mm, rotated rx 180 ry 20 rz -150.43 deg; joints [9.652, -57.083, 156.851, 27.216, -28.223, 13.113]
  MoveL 449 to (88.9, 914.4, 0) mm, rotated rx -180 ry 20 rz -150.43 deg; joints [12.268, -57.075, 156.352, 29.518, -27.584, 13.427]
  MoveL 450 to (1091.34, 914.4, 0) mm, rotated rx 0 ry 90 rz 29.57 deg; joints [18.115, -38.243, 110.051, 49.145, -77.868, -13.659]
  MoveL 451 to (1096.93, 923.88, 0) mm, rotated rx 0 ry 90 rz 29.57 deg; joints [17.68, -38.164, 109.84, 48.734, -77.678, -13.669]
  MoveL 452 to (1113.37, 952.5, 0) mm, rotated rx 0 ry 90 rz 29.57 deg; joints [16.378, -37.925, 109.198, 47.505, -77.101, -13.694]
  MoveL 453 to (1113.37, 889, 0) mm, rotated rx 0 ry 90 rz 29.57 deg; joints [18.803, -37.285, 107.501, 50.098, -77.006, -15.05]
  Set speed (60.0 mm/s)
  MoveL 454 to (1097.33, 860.38, 0) mm, rotated rx 0 ry 90 rz 29.57 deg; joints [20.091, -37.474, 107.998, 51.32, -77.537, -15.086]
  MoveL 455 to (1091.87, 850.9, 0) mm, rotated rx 0 ry 90 rz 29.57 deg; joints [20.522, -37.535, 108.16, 51.728, -77.712, -15.097]
  MoveL 456 to (88.9, 850.9, 0) mm, rotated rx 0 ry 60 rz 29.57 deg; joints [67.754, -12.875, 156.052, 118.503, -102.197, 54.32]
  MoveL 457 to (88.9, 889, 0) mm, rotated rx 0 ry 60 rz 29.57 deg; joints [66.314, -9.817, 157.3, 118.583, -101.18, 58.761]
  MoveL 458 to (1113.37, 889, 0) mm, rotated rx 0 ry 90 rz 29.57 deg; joints [18.803, -37.285, 107.501, 50.098, -77.006, -15.05]
  MoveL 459 to (1113.37, 825.5, 0) mm, rotated rx 0 ry 90 rz 29.57 deg; joints [21.159, -36.54, 105.554, 52.643, -76.898, -16.54]
  Set speed (60.0 mm/s)
  MoveL 460 to (88.9, 825.5, 0) mm, rotated rx 0 ry 60 rz 29.57 deg; joints [68.625, -14.747, 155.137, 118.423, -102.924, 51.476]
  MoveL 461 to (88.9, 787.4, 0) mm, rotated rx 0 ry 60 rz 29.57 deg; joints [69.816, -17.304, 153.65, 118.259, -104.061, 47.381]
  MoveL 462 to (1092.4, 787.4, 0) mm, rotated rx 0 ry 90 rz 29.57 deg; joints [22.855, -36.719, 106.02, 54.257, -77.553, -16.672]
  MoveL 463 to (1097.73, 796.89, 0) mm, rotated rx 0 ry 90 rz 29.57 deg; joints [22.43, -36.676, 105.906, 53.853, -77.39, -16.64]
  MoveL 464 to (1113.37, 825.5, 0) mm, rotated rx 0 ry 90 rz 29.57 deg; joints [21.159, -36.54, 105.554, 52.643, -76.898, -16.54]
  MoveL 465 to (1113.37, 762, 0) mm, rotated rx 0 ry 90 rz 29.57 deg; joints [23.443, -35.684, 103.354, 55.136, -76.787, -18.164]
  Set speed (60.0 mm/s)
  MoveL 466 to (1098.13, 733.39, 0) mm, rotated rx 0 ry 90 rz 29.57 deg; joints [24.691, -35.765, 103.561, 56.328, -77.248, -18.331]
  MoveL 467 to (1092.95, 723.9, 0) mm, rotated rx 0 ry 90 rz 29.57 deg; joints [25.107, -35.791, 103.626, 56.726, -77.401, -18.386]
  MoveL 468 to (88.9, 723.9, 0) mm, rotated rx 0 ry 70 rz 29.57 deg; joints [69.285, -28.239, 155.077, 109.063, -100.777, 37.089]
  MoveL 469 to (88.9, 762, 0) mm, rotated rx 0 ry 70 rz 29.57 deg; joints [68.162, -26.182, 156.903, 108.909, -100.179, 41.055]
  MoveL 470 to (1113.37, 762, 0) mm, rotated rx 0 ry 90 rz 29.57 deg; joints [23.443, -35.684, 103.354, 55.136, -76.787, -18.164]
  MoveL 471 to (1113.37, 698.5, 0) mm, rotated rx 0 ry 90 rz 29.57 deg; joints [25.651, -34.712, 100.898, 57.571, -76.685, -19.926]
  Set speed (60.0 mm/s)
  MoveL 472 to (88.9, 698.5, 0) mm, rotated rx 0 ry 80 rz 29.57 deg; joints [66.775, -36.977, 157.224, 100.506, -95.461, 30.193]
  MoveL 473 to (88.9, 660.4, 0) mm, rotated rx 0 ry 90 rz 29.57 deg; joints [63.931, -45.546, 157.635, 93.246, -88.684, 22.052]
  MoveL 474 to (1093.5, 660.4, 0) mm, rotated rx 0 ry 90 rz 29.57 deg; joints [27.279, -34.743, 100.974, 59.132, -77.268, -20.24]
  MoveL 475 to (1098.54, 669.89, 0) mm, rotated rx 0 ry 90 rz 29.57 deg; joints [26.872, -34.736, 100.958, 58.742, -77.122, -20.162]
  MoveL 476 to (1113.37, 698.5, 0) mm, rotated rx 0 ry 90 rz 29.57 deg; joints [25.651, -34.712, 100.898, 57.571, -76.685, -19.926]
  MoveL 477 to (1113.37, 635, 0) mm, rotated rx 0 ry 90 rz 29.57 deg; joints [27.779, -33.618, 98.178, 59.946, -76.6, -21.827]
  Set speed (60.0 mm/s)
  MoveL 478 to (1098.95, 606.38, 0) mm, rotated rx 0 ry 90 rz 29.57 deg; joints [28.97, -33.582, 98.09, 61.091, -77.02, -22.133]
  MoveL 479 to (1094.06, 596.9, 0) mm, rotated rx 0 ry 90 rz 29.57 deg; joints [29.366, -33.568, 98.056, 61.471, -77.16, -22.235]
  MoveL 480 to (88.9, 596.9, 0) mm, rotated rx 0 ry 90 rz 29.57 deg; joints [65.86, -46.697, 153.912, 95.19, -88.395, 17.142]
  MoveL 481 to (88.9, 635, 0) mm, rotated rx 0 ry 90 rz 29.57 deg; joints [64.736, -46.087, 156.167, 94.047, -88.522, 20.028]
  MoveL 482 to (1113.37, 635, 0) mm, rotated rx 0 ry 90 rz 29.57 deg; joints [27.779, -33.618, 98.178, 59.946, -76.6, -21.827]
  MoveL 483 to (88.9, 317.5, 0) mm, rotated rx 0 ry 90 rz 29.57 deg; joints [71.879, -46.015, 135.702, 101.45, -90.062, -0.307]
  Set speed (60.0 mm/s)
  MoveL 484 to (88.9, 279.4, 0) mm, rotated rx 0 ry 90 rz 29.57 deg; joints [72.482, -45.43, 133.007, 102.043, -90.506, -2.369]
  MoveL 485 to (1098.24, 279.4, 0) mm, rotated rx 0 ry 90 rz 29.57 deg; joints [38.535, -25.357, 78.734, 72.124, -77.147, -34.593]
  MoveL 486 to (1102.05, 288.92, 0) mm, rotated rx 0 ry 90 rz 29.57 deg; joints [38.208, -25.51, 79.082, 71.805, -77.023, -34.341]
  MoveL 487 to (1113.37, 317.5, 0) mm, rotated rx 0 ry 90 rz 29.57 deg; joints [37.222, -25.953, 80.089, 70.84, -76.653, -33.601]
  MoveL 488 to (88.9, 317.5, 0) mm, rotated rx 0 ry 90 rz 29.57 deg; joints [71.879, -46.015, 135.702, 101.45, -90.062, -0.307]
  MoveL 489 to (88.9, 254, 0) mm, rotated rx 0 ry 90 rz 29.57 deg; joints [72.863, -44.992, 131.182, 102.408, -90.82, -3.721]
  Set speed (60.0 mm/s)
  MoveL 490 to (1113.37, 254, 0) mm, rotated rx 0 ry 90 rz 29.57 deg; joints [38.877, -23.86, 75.355, 72.825, -76.78, -36.499]
  MoveL 491 to (1102.52, 225.42, 0) mm, rotated rx 0 ry 90 rz 29.57 deg; joints [39.822, -23.313, 74.131, 73.751, -77.152, -37.341]
  MoveL 492 to (1098.88, 215.9, 0) mm, rotated rx 0 ry 90 rz 29.57 deg; joints [40.135, -23.124, 73.706, 74.057, -77.278, -37.629]
  MoveL 493 to (88.9, 215.9, 0) mm, rotated rx 0 ry 90 rz 29.57 deg; joints [73.405, -44.265, 128.399, 102.911, -91.315, -5.718]
  MoveL 494 to (88.9, 254, 0) mm, rotated rx 0 ry 90 rz 29.57 deg; joints [72.863, -44.992, 131.182, 102.408, -90.82, -3.721]
  MoveL 495 to (88.9, 190.5, 0) mm, rotated rx 0 ry 90 rz 29.57 deg; joints [73.748, -43.737, 126.512, 103.217, -91.66, -7.033]
  Set speed (60.0 mm/s)
  MoveL 496 to (88.9, 152.4, 0) mm, rotated rx 0 ry 90 rz 29.57 deg; joints [74.238, -42.883, 123.634, 103.636, -92.199, -8.986]
  MoveL 497 to (1099.53, 152.4, 0) mm, rotated rx 0 ry 90 rz 29.57 deg; joints [41.662, -20.601, 68.108, 75.935, -77.448, -40.939]
  MoveL 498 to (1102.99, 161.93, 0) mm, rotated rx 0 ry 90 rz 29.57 deg; joints [41.363, -20.835, 68.623, 75.642, -77.322, -40.609]
  MoveL 499 to (1113.37, 190.5, 0) mm, rotated rx 0 ry 90 rz 29.57 deg; joints [40.458, -21.505, 70.104, 74.753, -76.946, -39.646]
  MoveL 500 to (88.9, 190.5, 0) mm, rotated rx 0 ry 90 rz 29.57 deg; joints [73.748, -43.737, 126.512, 103.217, -91.66, -7.033]
  MoveL 501 to (88.9, 127, 0) mm, rotated rx 0 ry 90 rz 29.57 deg; joints [74.548, -42.274, 121.682, 103.889, -92.57, -10.279]
  Set speed (60.0 mm/s)
  MoveL 502 to (1113.37, 127, 0) mm, rotated rx 0 ry 90 rz 29.57 deg; joints [41.967, -18.821, 64.202, 76.633, -77.149, -43.107]
  MoveL 503 to (1104.01, 98.53, 0) mm, rotated rx 0 ry 90 rz 29.57 deg; joints [42.819, -17.973, 62.353, 77.483, -77.513, -44.245]
  MoveL 504 to (1100.86, 88.9, 0) mm, rotated rx 0 ry 90 rz 29.57 deg; joints [43.104, -17.672, 61.697, 77.768, -77.636, -44.644]
  MoveL 505 to (88.9, 88.9, 0) mm, rotated rx 0 ry 90 rz 29.57 deg; joints [74.993, -41.301, 118.7, 104.228, -93.145, -12.209]
  MoveL 506 to (88.9, 127, 0) mm, rotated rx 0 ry 90 rz 29.57 deg; joints [74.548, -42.274, 121.682, 103.889, -92.57, -10.279]
  MoveL 507 to (88.9, 63.5, 0) mm, rotated rx 0 ry 90 rz 29.57 deg; joints [75.275, -40.614, 116.674, 104.428, -93.539, -13.492]
  Set speed (60.0 mm/s)
  MoveL 508 to (88.9, 25.4, 0) mm, rotated rx 0 ry 90 rz 29.57 deg; joints [75.68, -39.527, 113.575, 104.69, -94.146, -15.417]
  MoveL 509 to (1101.55, 25.4, 0) mm, rotated rx 0 ry 90 rz 29.57 deg; joints [44.492, -14.252, 54.319, 79.585, -77.87, -48.823]
  MoveL 510 to (1104.5, 35.01, 0) mm, rotated rx 0 ry 90 rz 29.57 deg; joints [44.221, -14.633, 55.137, 79.309, -77.747, -48.345]
  MoveL 511 to (1113.37, 63.5, 0) mm, rotated rx 0 ry 90 rz 29.57 deg; joints [43.409, -15.698, 57.427, 78.484, -77.382, -46.994]
  MoveL 512 to (88.9, 63.5, 0) mm, rotated rx 0 ry 90 rz 29.57 deg; joints [75.275, -40.614, 116.674, 104.428, -93.539, -13.492]
  MoveL 513 to (181.97, 1023.42, 0) mm, rotated rx 0 ry 50 rz 29.57 deg; joints [52.096, 2.597, 153.85, 125.711, -111.016, 76.323]
  Set speed (60.0 mm/s)
  MoveL 514 to (213.62, 1020.12, 0) mm, rotated rx 0 ry 50 rz 29.57 deg; joints [49.605, 0.497, 153.338, 124.312, -114.365, 75.411]
